// TwinCAT 3 PLC project PLC_PlantControl
// Title: PlantControl and CMs
// Company: ArmAutomation
// ProjectVersion: 0.1.0.0
// Description: This library hold functionality for a control structure and Control modules
// ProgramVersion: 3.1.4024.0
// libraries:
//   Tc2_ControllerToolbox, * (Beckhoff Automation GmbH)
//   Tc2_Standard, * (Beckhoff Automation GmbH)
//   Tc2_System, * (Beckhoff Automation GmbH)
//   Tc3_Module, * (Beckhoff Automation GmbH)
// project tree:
//   DUTs/Control Function UDTs/ ENUM_MODE_HANDLER.TcDUT
//   DUTs/V1/ Udt_CM_Actuator2State.TcDUT, Udt_CM_Actuator3State.TcDUT (not stored), Udt_CM_ActuatorAnalog.TcDUT (not stored), Udt_CM_Sensor2State.TcDUT, Udt_CM_SensorAnalog.TcDUT, Udt_PlantControl.TcDUT, Udt_PlantControl_SCADA.TcDUT (not stored)
//   DUTs/V2/ Udt_CM_Actuator2State_V2.TcDUT, Udt_CM_AO_V2.TcDUT, Udt_CM_Actuator3State_V2.TcDUT
//   GVLs/ FIO.TcGVL, OPC.TcGVL
//   / PlcTask.TcTTO
//   POUs/CM/ CM_Actuator2State.TcPOU, CM_Actuator3State.TcPOU, CM_ActuatorAnalog.TcPOU, CM_Sensor2State.TcPOU, CM_SensorAnalog.TcPOU
//   POUs/CM_V2/ CM_Actuator2State_V2.TcPOU, CM_Actuator3State_V2.TcPOU, CM_AO_V2.TcPOU, CM_Sensor2State_V2.TcPOU, CM_SensorAnalog_V2.TcPOU
//   POUs/Control functions/ FB_MODE_HANDLER.TcPOU, FB_PID.TcPOU
//   POUs/EM/ EM_Tank.TcPOU
//   POUs/ MAIN.TcPOU
//   POUs/Plant Control/ FB_PlantControl.TcPOU, FB_PlantControl_V2.TcPOU
//   POUs/Scaling/ FB_ScaleIN_1.TcPOU, FB_ScaleOut_1.TcPOU
//   POUs/System/ FB_ScaleIN.TcPOU, FB_ScaleOut.TcPOU, systemTimeDelay.TcPOU, SystemTimeTick.TcPOU
//   Version/ Global_Version.TcGVL
// real-time tasks:
//   TASK PlcTask: cycle T#10ms, priority 20, ADS port 350

CONFIGURATION PLC_PlantControl
    RESOURCE PLC ON TwinCAT3
        TASK PlcTask(INTERVAL := T#10ms, PRIORITY := 20);
        PROGRAM MAIN WITH PlcTask : MAIN;
    END_RESOURCE
END_CONFIGURATION

// ---- DUTs/Control Function UDTs/ENUM_MODE_HANDLER.TcDUT
{attribute 'qualified_only'}
{attribute 'strict'}
TYPE ENUM_MODE_HANDLER :
(
    MODE_EMGSTOP := 0,
    MODE_AUTO := 1,
    MODE_MAN  := 2
);
END_TYPE

// ---- DUTs/V1/Udt_CM_Actuator2State.TcDUT
TYPE Udt_CM_Actuator2State :
STRUCT
	PI_MANUAL :BOOL;
	PI_AUTO : BOOL;
	PI_HMI_HAND : BOOL;
	
	PI_AlarmHigh_Enable : BOOL;
	PI_AlarmLow_Enable : BOOL;
	
	PI_Alarm_Ack_H : BOOL;
	PI_Alarm_Ack_L : BOOL;
	
	PI_Interlock : BOOL;
	PO_Interlocked : BOOL;
	
	PO_ALARM_H : BOOL;
	PO_ALARM_L : BOOL;
	
	PO_HMI_HAND_ON: BOOL;
	PO_AUTO_ON : BOOL;
	PO_MANUAL_ON : BOOL;
	PO_ON : BOOL;
	PO_OFF :BOOL;
	
	
END_STRUCT
END_TYPE

// ---- DUTs/V1/Udt_CM_Sensor2State.TcDUT
TYPE Udt_CM_Sensor2State :
STRUCT
	PI_ManualMode : BOOL;
	PI_AutoHigh : BOOL;
	
	PI_HMI_HAND : BOOL;
	PI_HMI_HAND_ON : BOOL;
	
	PI_AlarmHighEnable : BOOL;
	PI_AlarmLowEnable : BOOL;
	
	PI_Alarmdelay_H : INT;
	PI_Alarmdelay_L : INT;
	
	PO_Alarm_H : BOOL;
	PO_Alarm_L : BOOL;
	
	PO_HMI_HAND : BOOL;
	PO_High : BOOL;
	
	PO_HIST_BIT_H : BOOL;
	PO_HIST_BIT_L : BOOL;

END_STRUCT
END_TYPE

// ---- DUTs/V1/Udt_CM_SensorAnalog.TcDUT
TYPE Udt_CM_SensorAnalog :
STRUCT
	PI_ManualMode : BOOL;
	PI_AutoMode : BOOL;
	
	PI_AlarmHighEnable : BOOL;
	PI_AlarmLowEnable : BOOL;
	PI_AlarmHighHighEnable : BOOL;
	PI_AlarmLowLowEnable : BOOL;
	
	PI_Alarm_Ack_HH : BOOL;
	PI_Alarm_Ack_H : BOOL;
	PI_Alarm_Ack_L : BOOL;
	PI_Alarm_Ack_LL : BOOL;
	
	
	PI_PV :INT;
	PI_PV_REAL : REAL;
	
	PI_PV_MAX : INT;
	PI_PV_MIN : INT;

	
	PO_PV_REAL : REAL;
	PO_PV_SCALED : REAL;
	
	
	PO_ALARM_HH : BOOL;
	PO_ALARM_H : BOOL;
	PO_ALARM_L : BOOL;
	PO_ALARM_LL : BOOL;
	
	PO_HIST_BIT_HH : BOOL;
	PO_HIST_BIT_H : BOOL;
	PO_HIST_BIT_L : BOOL;
	PO_HIST_BIT_LL : BOOL;
	
	
END_STRUCT
END_TYPE

// ---- DUTs/V1/Udt_PlantControl.TcDUT
TYPE Udt_PlantControl :
STRUCT
	
	PI_Auto : BOOL;
	PI_Manual : BOOL;
	
	
	PI_Start : BOOL;
	PI_Stop : BOOL := TRUE;
	PI_Reset : BOOL;
	PI_ResetEmgStop_5s :BOOL;
	
	PI_EmgStop : BOOL := TRUE;
	
	PO_Manual : BOOL;
	
	
	PO_Auto : BOOL;
	PO_Startet : BOOL;
	PO_Stopped : BOOL;
	PO_Reset : BOOL;
	PO_ResetEmgStop_5s :BOOL;
	
	PO_EmgStopped : BOOL;
	
	PO_ON : BOOL;
	
	PO_MODE : ENUM_MODE_HANDLER;
END_STRUCT
END_TYPE

// ---- DUTs/V2/Udt_CM_Actuator2State_V2.TcDUT
TYPE Udt_CM_Actuator2State_V2 :
STRUCT
	PI_MANUAL :BOOL;
	PI_AUTO : BOOL;
	PI_HMI_HAND : BOOL;
	
	PI_AlarmHigh_Enable : BOOL;
	PI_AlarmLow_Enable : BOOL;
	
	PI_Alarm_Condition_H : BOOL;
	PI_Alarm_Condition_L : BOOL;
	
	PI_AlarmDelay_H : LREAL;
	PI_AlarmDelay_L : LREAL;
	
	PI_Alarm_Ack_H : BOOL;
	PI_Alarm_Ack_L : BOOL;
	
	PI_Interlock : BOOL;
	(*PO_Interlocked : BOOL;
	
	PO_ALARM_H : BOOL;
	PO_ALARM_L : BOOL;
	
	PO_HMI_HAND_ON: BOOL;
	PO_AUTO_ON : BOOL;
	PO_MANUAL_ON : BOOL;
	PO_ON : BOOL;
	PO_OFF :BOOL;
	*)
	
	PO_MODE : ENUM_MODE_HANDLER;
	
END_STRUCT
END_TYPE

// ---- DUTs/V2/Udt_CM_AO_V2.TcDUT
TYPE Udt_CM_AO_V2 :
STRUCT
	PI_MANUAL :BOOL;
	PI_AUTO : BOOL;
	PI_HMI_HAND : BOOL; 
	
	PI_MANUAL_ON_1 : BOOL;
	PI_MANUAL_ON_2 : BOOL;
	
	PI_AUTO_ON_1 : BOOL;
	PI_AUTO_ON_2 : BOOL;
	
	PI_INTERLOCK : BOOL;
	
	PI_OFF : BOOL;
	
	PO_HMI_HAND_ON : BOOL;
	PO_AUTO_ON : BOOL;
	PO_ON : BOOL;
	
	
	PO_INTERLOCKED : BOOL;
	
	PO_OUT_OFF :BOOL;
	
	PI_Alarm_Ack_HH : BOOL;
	PI_Alarm_Ack_H : BOOL;
	PI_Alarm_Ack_L : BOOL;
	PI_Alarm_Ack_LL : BOOL;
	
	PO_MODE : ENUM_MODE_HANDLER;
END_STRUCT
END_TYPE

// ---- DUTs/V2/Udt_CM_Actuator3State_V2.TcDUT
TYPE Udt_CM_Actuator3State_V2 :
STRUCT
	PI_MANUAL :BOOL;
	PI_HMI_HAND : BOOL;
	PI_AUTO : BOOL;
	
	PI_MANUAL_ON_1 : BOOL;
	PI_MANUAL_ON_2 : BOOL;
	
	PI_AUTO_ON_1 : BOOL;
	PI_AUTO_ON_2 : BOOL;
	
	PI_OFF : BOOL;
	
	PI_Alarm_Enable : BOOL;
	PI_CM_Alarm : BOOL;
	
	PI_CM_Interlock : BOOL;
	
	PO_AUTO_ON :BOOL;
	PO_MANUAL_ON :BOOL;
	PO_HMI_HAND_ON : BOOL;
	
	PO_ON_1 : BOOL;
	PO_ON_2 : BOOL;
	
	PO_OFF :BOOL;
	
	PO_CM_Alarm : BOOL;
	
	PO_CM_Interlocked : BOOL;
	
	PO_MODE : ENUM_MODE_HANDLER;


END_STRUCT
END_TYPE

// ---- GVLs/FIO.TcGVL
{attribute 'qualified_only'}
VAR_GLOBAL
	
	(*bEmgStop : BOOL := TRUE; //Sensor	Bool	Emergency stop	0	TRUE
	bStart : BOOL;	//Sensor	Bool	Start	1	FALSE
	bStop : BOOL := TRUE;	//Sensor	Bool	Stop	3	TRUE
	bReset : BOOL;	//Sensor	Bool	Reset	4	FALSE
	bManual : BOOL;	//Sensor	Bool	Manual	5	TRUE
	bAuto : BOOL; 	//Sensor	Bool	Auto	6	FALSE
	
	bGreenLight : BOOL;
	bYellowLight : BOOL;
	bRedLight : BOOL;*)
		
	Plant_control : Udt_PlantControl;
	
END_VAR

// ---- GVLs/OPC.TcGVL
{attribute 'qualified_only'}
VAR_GLOBAL
	//cmActuator2State : Udt_CM_Actuator2State;
	Udt_PlantControl : Udt_PlantControl;
	
	Plant_1_Control : Udt_PlantControl;
END_VAR

// ---- Version/Global_Version.TcGVL
{attribute 'TcGenerated'}
{attribute 'no-analysis'}
{attribute 'linkalways'}
// This function has been automatically generated from the project information.
VAR_GLOBAL CONSTANT
	{attribute 'const_non_replaced'}
	stLibVersion_PlantControl_and_CMs : ST_LibVersion := (iMajor := 0, iMinor := 1, iBuild := 0, iRevision := 0, nFlags := 0, sVersion := '0.1.0.0');
END_VAR

// ---- POUs/MAIN.TcPOU
PROGRAM MAIN
VAR
	//Plant_Control : FB_PlantControl;
END_VAR
VAR_IN_OUT
	
END_VAR


(*fbPlantControl(
		//Set up variables to IO here
		
		(*Auto_In := HMI.bAuto,
		Manual_In := HMI.bManual,
		
		
		Start_In := HMI.bStart,
		Stop_In := HMI.bStop,
		EmgStop_In := HMI.bEmgStop,
		Reset_In := HMI.bReset,
		
		Startet_Out => HMI.bGreenLight,
		Stopped_Out => HMI.bYellowLight,
		EmgStopped_Out => HMI.bRedLight,*)
	
		Ctrl_Plant := FIO.Plant_control
		);
	
cmActuator2State(
	CM_UDT_CTRL := OPC.cmActuator2State,
	Plant_control := FIO.Plant_control
	);
	
	*)

END_PROGRAM

// ---- POUs/CM/CM_Actuator2State.TcPOU
FUNCTION_BLOCK CM_Actuator2State
VAR_INPUT
	CM_Number : INT;
	
	PI_MANUAL :BOOL;
	PI_AUTO : BOOL;
	
	PI_HMI_HAND : BOOL;
	
	PI_MANUAL_ON : BOOL;
	PI_AUTO_ON : BOOL;
	
	PI_OFF : BOOL;
	
	PI_AlarmHigh_Enable : BOOL;
	PI_AlarmLow_Enable : BOOL;
	PI_AlarmDelay_H : ULINT;
	PI_AlarmDelay_L : ULINT;
	
	PI_Alarm_Condition_H : BOOL;
	PI_Alarm_Condition_L : BOOL;
	
	PI_CM_Interlock : BOOL;
	
END_VAR
VAR_OUTPUT
	
	PO_AUTO_ON :BOOL;
	PO_MANUAL_ON : BOOL;
	PO_HMI_HAND_ON : BOOL;
	
	PO_OUT_ON : BOOL;
	OUT_OFF :BOOL;
	
	
	PO_ALARM_H : BOOL;
	PO_ALARM_L : BOOL;;
	
	PO_Interlocked : BOOL;
	
END_VAR
VAR
	SR_Auto: SR;
	SR_Manual : SR;
	
	Alarm_limit_Exceeded_H : BOOL;
	Alarm_limit_Exceeded_L : BOOL;
	
	Alarm_Ack_H : BOOL;
	Alarm_Ack_L : BOOL;
	
	alarmDelay_H : systemTimeDelay;
	alarmDelay_L : systemTimeDelay;
END_VAR
VAR_IN_OUT
	CM_UDT_CTRL : Udt_CM_Actuator2State;
END_VAR
VAR // added by the converter: edge detectors and wires of the graphical bodies
    _w1 : BOOL;
END_VAR

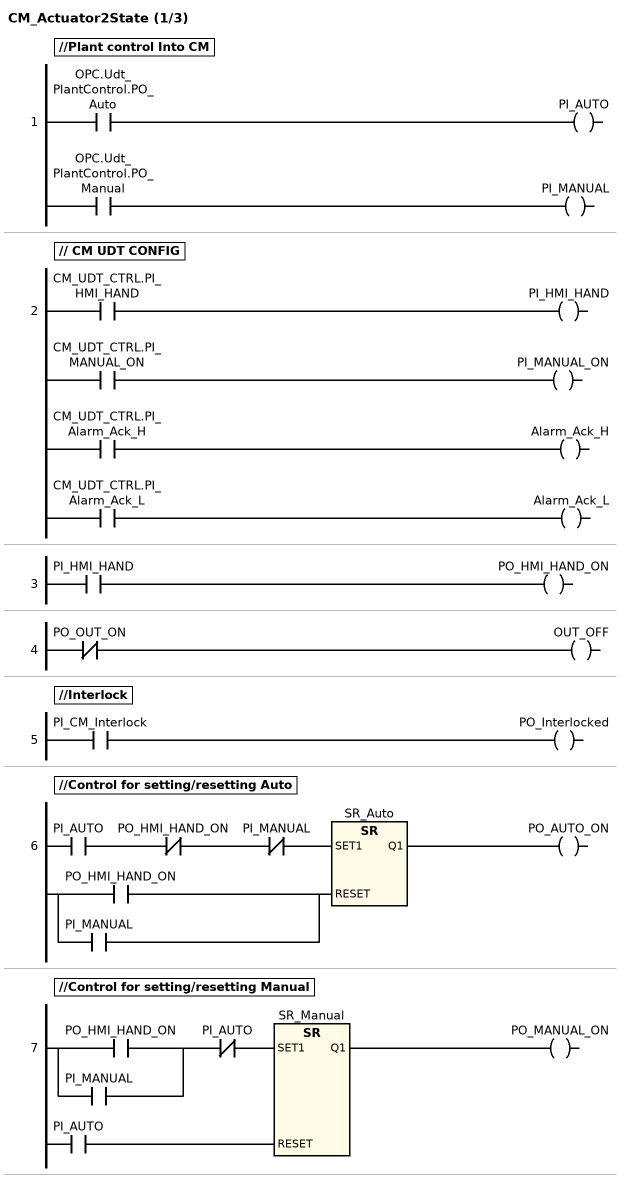
// NETWORK 1
// label: //Plant control Into CM
PI_AUTO := OPC.Udt_PlantControl.PO_Auto;
PI_MANUAL := OPC.Udt_PlantControl.PO_Manual;

// NETWORK 2
// label: // CM UDT CONFIG
PI_HMI_HAND := CM_UDT_CTRL.PI_HMI_HAND;
PI_MANUAL_ON := CM_UDT_CTRL.PI_MANUAL_ON;
Alarm_Ack_H := CM_UDT_CTRL.PI_Alarm_Ack_H;
Alarm_Ack_L := CM_UDT_CTRL.PI_Alarm_Ack_L;

// NETWORK 3
PO_HMI_HAND_ON := PI_HMI_HAND;

// NETWORK 4
OUT_OFF := NOT PO_OUT_ON;

// NETWORK 5
// label: //Interlock
PO_Interlocked := PI_CM_Interlock;

// NETWORK 6
// label: //Control for setting/resetting Auto
SR_Auto(SET1 := PI_AUTO AND NOT PO_HMI_HAND_ON AND NOT PI_MANUAL, RESET := PO_HMI_HAND_ON OR PI_MANUAL); // SR
PO_AUTO_ON := SR_Auto.Q1;

// NETWORK 7
// label: //Control for setting/resetting Manual
SR_Manual(SET1 := (PO_HMI_HAND_ON OR PI_MANUAL) AND NOT PI_AUTO, RESET := PI_AUTO); // SR
PO_MANUAL_ON := SR_Manual.Q1;

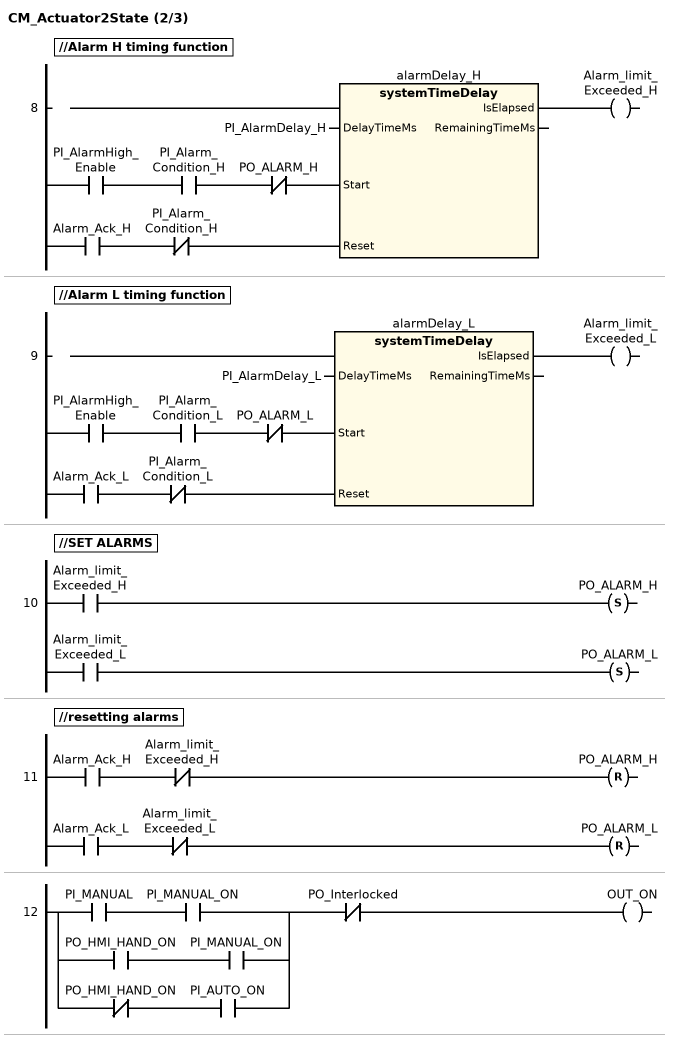
// NETWORK 8
// label: //Alarm H timing function
alarmDelay_H(
    DelayTimeMs := PI_AlarmDelay_H,
    Start := PI_AlarmHigh_Enable AND PI_Alarm_Condition_H AND NOT PO_ALARM_H,
    Reset := Alarm_Ack_H AND NOT PI_Alarm_Condition_H); // systemTimeDelay
Alarm_limit_Exceeded_H := alarmDelay_H.IsElapsed;

// NETWORK 9
// label: //Alarm L timing function
alarmDelay_L(
    DelayTimeMs := PI_AlarmDelay_L,
    Start := PI_AlarmHigh_Enable AND PI_Alarm_Condition_L AND NOT PO_ALARM_L,
    Reset := Alarm_Ack_L AND NOT PI_Alarm_Condition_L); // systemTimeDelay
Alarm_limit_Exceeded_L := alarmDelay_L.IsElapsed;

// NETWORK 10
// label: //SET ALARMS
PO_ALARM_H S= Alarm_limit_Exceeded_H;
PO_ALARM_L S= Alarm_limit_Exceeded_L;

// NETWORK 11
// label: //resetting alarms
PO_ALARM_H R= Alarm_Ack_H AND NOT Alarm_limit_Exceeded_H;
PO_ALARM_L R= Alarm_Ack_L AND NOT Alarm_limit_Exceeded_L;

// NETWORK 12
OUT_ON := (PI_MANUAL AND PI_MANUAL_ON OR PO_HMI_HAND_ON AND PI_MANUAL_ON OR NOT PO_HMI_HAND_ON AND PI_AUTO_ON) AND NOT PO_Interlocked;

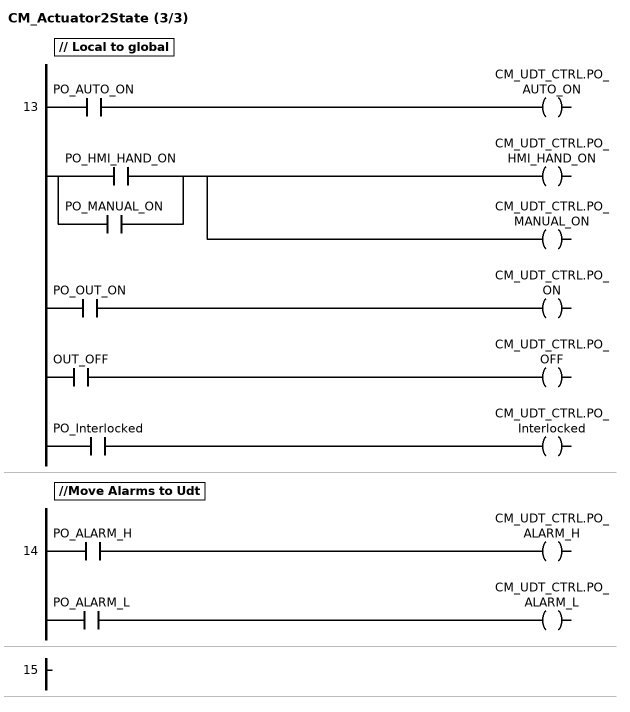
// NETWORK 13
// label: // Local to global
CM_UDT_CTRL.PO_AUTO_ON := PO_AUTO_ON;
_w1 := PO_HMI_HAND_ON OR PO_MANUAL_ON;
CM_UDT_CTRL.PO_HMI_HAND_ON := _w1;
CM_UDT_CTRL.PO_MANUAL_ON := _w1;
CM_UDT_CTRL.PO_ON := PO_OUT_ON;
CM_UDT_CTRL.PO_OFF := OUT_OFF;
CM_UDT_CTRL.PO_Interlocked := PO_Interlocked;

// NETWORK 14
// label: //Move Alarms to Udt
CM_UDT_CTRL.PO_ALARM_H := PO_ALARM_H;
CM_UDT_CTRL.PO_ALARM_L := PO_ALARM_L;

// NETWORK 15

END_FUNCTION_BLOCK

// ---- POUs/System/systemTimeDelay.TcPOU
FUNCTION_BLOCK systemTimeDelay
VAR_INPUT
    DelayTime : LREAL;   // Desired delay in seconds
    Start     : BOOL;    // Start signal (must stay TRUE to complete delay)
    Reset     : BOOL;    // Resets latched state and timer
END_VAR

VAR_OUTPUT
    IsElapsed     : BOOL;    // Latches TRUE after timeout, until reset
    RemainingTime : LREAL;   // Countdown in seconds (0 if not running)
END_VAR

VAR
    StartEdge       : BOOL;
    PrevStart       : BOOL;
    StartTime       : ULINT;   // Time when timer started (µs)
    ElapsedTimeRaw  : ULINT;   // Raw elapsed time in microseconds
    ElapsedSeconds  : LREAL;   // Elapsed time in seconds
    IsRunning       : BOOL;
END_VAR

// Detect rising edge of Start
StartEdge := Start AND NOT PrevStart;
PrevStart := Start;

// Reset everything if Reset = TRUE
IF Reset THEN
    IsElapsed := FALSE;
    IsRunning := FALSE;
    RemainingTime := 0.0;
END_IF

// If Start goes low during active timing, cancel and reset
IF NOT Start AND IsRunning THEN
    IsRunning := FALSE;
    RemainingTime := 0.0;
END_IF

// Start timer on rising edge of Start
IF StartEdge AND NOT IsElapsed THEN
    StartTime := F_GetSystemTime();  // System time in microseconds
    IsRunning := TRUE;
END_IF

// Timing logic
IF IsRunning THEN
    ElapsedTimeRaw := F_GetSystemTime() - StartTime;       // Time difference in µs
    ElapsedSeconds := ElapsedTimeRaw / 10000000.0;          // Convert to seconds

    IF ElapsedSeconds >= DelayTime THEN
        IsElapsed := TRUE;
        IsRunning := FALSE;
        RemainingTime := 0.0;
    ELSE
        RemainingTime := DelayTime - ElapsedSeconds;
    END_IF
END_IF

END_FUNCTION_BLOCK

// ---- POUs/CM/CM_Actuator3State.TcPOU
FUNCTION_BLOCK CM_Actuator3State
VAR_INPUT
	CM_Number : INT;
	
	IN_MANUAL :BOOL;
	IN_HMI_HAND : BOOL;
	IN_AUTO : BOOL;
	
	IN_MANUAL_ON_1 : BOOL;
	IN_MANUAL_ON_2 : BOOL;
	
	IN_AUTO_ON_1 : BOOL;
	IN_AUTO_ON_2 : BOOL;
	
	IN_OFF : BOOL;
	
	IN_Alarm_Enable : BOOL;
	IN_CM_Alarm : BOOL;
	
	IN_CM_Interlock : BOOL;
END_VAR
VAR_OUTPUT
	AUTO_ON :BOOL;
	HMI_HAND_ON : BOOL;
	
	OUT_ON_1 : BOOL;
	OUT_ON_2 : BOOL;
	
	OUT_OFF :BOOL;
	
	PO_CM_Alarm : BOOL;
	
	PO_CM_Interlocked : BOOL;
END_VAR
VAR
	alarmDelay_H : systemTimeDelay;
	alarmDelay_L : systemTimeDelay;
END_VAR
VAR_IN_OUT
	CM_UDT_CTRL : Udt_CM_Actuator3State;
	Plant_control : Udt_PlantControl;
END_VAR

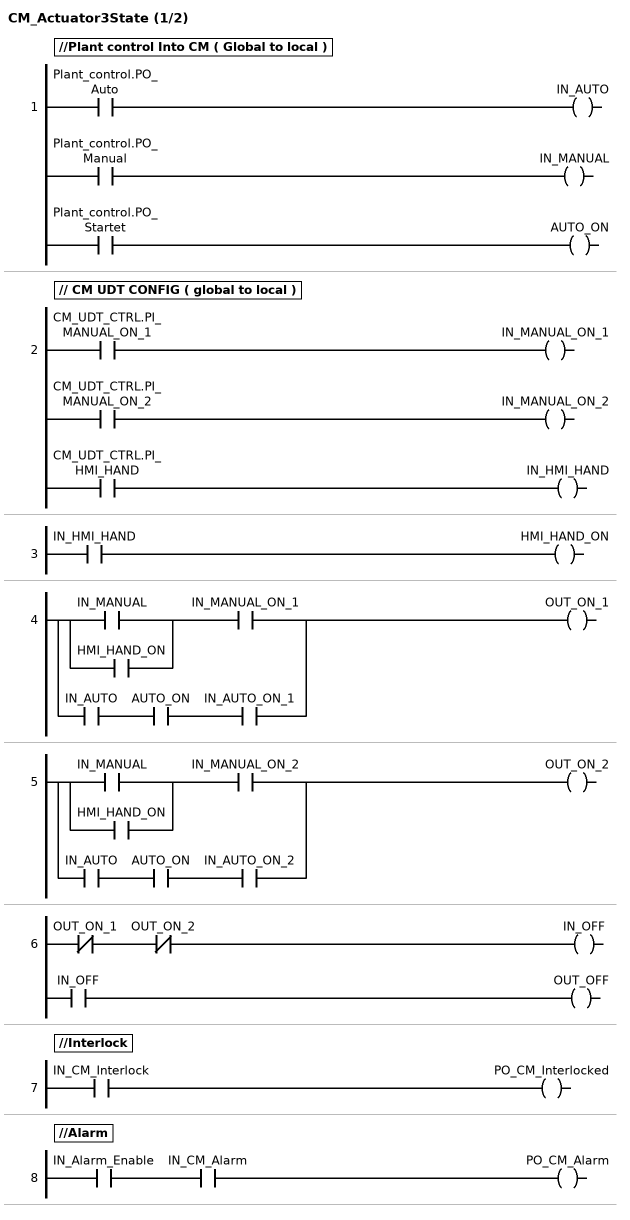
// NETWORK 1
// label: //Plant control Into CM ( Global to local )
IN_AUTO := Plant_control.PO_Auto;
IN_MANUAL := Plant_control.PO_Manual;
AUTO_ON := Plant_control.PO_Startet;

// NETWORK 2
// label: // CM UDT CONFIG ( global to local )
IN_MANUAL_ON_1 := CM_UDT_CTRL.PI_MANUAL_ON_1;
IN_MANUAL_ON_2 := CM_UDT_CTRL.PI_MANUAL_ON_2;
IN_HMI_HAND := CM_UDT_CTRL.PI_HMI_HAND;

// NETWORK 3
HMI_HAND_ON := IN_HMI_HAND;

// NETWORK 4
OUT_ON_1 := (IN_MANUAL OR HMI_HAND_ON) AND IN_MANUAL_ON_1 OR IN_AUTO AND AUTO_ON AND IN_AUTO_ON_1;

// NETWORK 5
OUT_ON_2 := (IN_MANUAL OR HMI_HAND_ON) AND IN_MANUAL_ON_2 OR IN_AUTO AND AUTO_ON AND IN_AUTO_ON_2;

// NETWORK 6
IN_OFF := NOT OUT_ON_1 AND NOT OUT_ON_2;
OUT_OFF := IN_OFF;

// NETWORK 7
// label: //Interlock
PO_CM_Interlocked := IN_CM_Interlock;

// NETWORK 8
// label: //Alarm
PO_CM_Alarm := IN_Alarm_Enable AND IN_CM_Alarm;

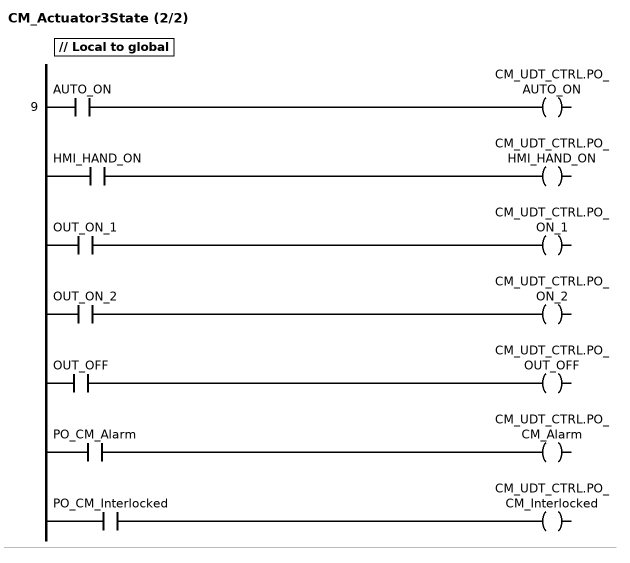
// NETWORK 9
// label: // Local to global
CM_UDT_CTRL.PO_AUTO_ON := AUTO_ON;
CM_UDT_CTRL.PO_HMI_HAND_ON := HMI_HAND_ON;
CM_UDT_CTRL.PO_ON_1 := OUT_ON_1;
CM_UDT_CTRL.PO_ON_2 := OUT_ON_2;
CM_UDT_CTRL.PO_OUT_OFF := OUT_OFF;
CM_UDT_CTRL.PO_CM_Alarm := PO_CM_Alarm;
CM_UDT_CTRL.PO_CM_Interlocked := PO_CM_Interlocked;

END_FUNCTION_BLOCK

// ---- POUs/CM/CM_ActuatorAnalog.TcPOU
FUNCTION_BLOCK CM_ActuatorAnalog
VAR_INPUT
	IN_MANUAL : BOOL;
	IN_AUTO : BOOL;
	IN_HMI_HAND : BOOL;
	
	IN_ON : BOOL;
	IN_OFF : BOOL;
	IN_EMG_STOP : BOOL;
	
	IN_RESET : BOOL;
	
	Input_analog : REAL;
	
	PV : REAL;
END_VAR
VAR_OUTPUT
	HMI_HAND_ON : BOOL;
	output_analog : REAL;
	Output_FB : BOOL;
END_VAR
VAR_IN_OUT
	CM_UDT_CTRL : Udt_CM_ActuatorAnalog;
	Plant_control : Udt_PlantControl;
END_VAR
VAR // added by the converter: edge detectors and wires of the graphical bodies
    _w1 : BOOL;
END_VAR

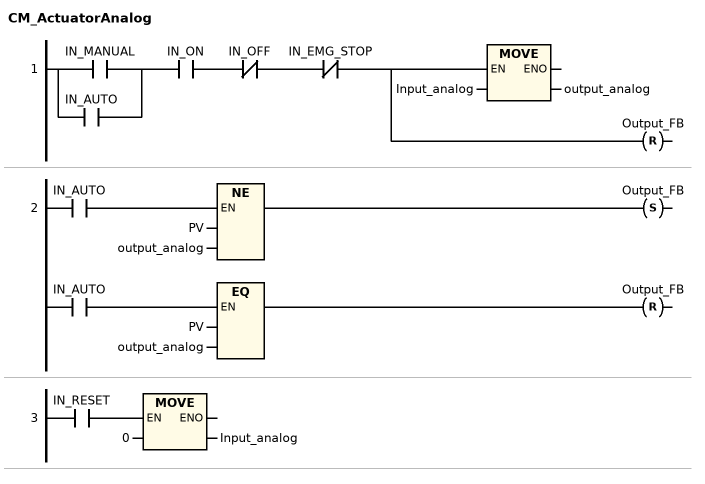
// NETWORK 1
_w1 := (IN_MANUAL OR IN_AUTO) AND IN_ON AND NOT IN_OFF AND NOT IN_EMG_STOP;
IF _w1 THEN output_analog := Input_analog; END_IF
Output_FB R= _w1;

// NETWORK 2
Output_FB S= IN_AUTO AND PV <> output_analog;
Output_FB R= IN_AUTO AND PV = output_analog;

// NETWORK 3
IF IN_RESET THEN Input_analog := 0; END_IF

END_FUNCTION_BLOCK

// ---- POUs/CM/CM_Sensor2State.TcPOU
FUNCTION_BLOCK CM_Sensor2State
VAR_INPUT
	PI_ManualMode : BOOL;
	PI_AutoMode : BOOL;
	
	PI_HMI_HAND : BOOL;
	PI_HMI_HAND_ON : BOOL;
	
	PI_Manual_ON : BOOL;
	PI_AutoHigh : BOOL;
	
	PI_AlarmHighEnable : BOOL;
	PI_AlarmLowEnable : BOOL;
	PI_Alarmdelay_H : DINT;
	PI_Alarmdelay_L : DINT;
	
	PI_Alarm_Condition_H : BOOL;
	PI_Alarm_Condition_L : BOOL;
	
	
	
END_VAR
VAR_OUTPUT
	PO_HMI_HAND : BOOL;
	PO_Manual : BOOL;
	PO_High : BOOL;
	
	PO_Alarm_H : BOOL;
	PO_Alarm_L : BOOL;
END_VAR
VAR
	Alarm_limit_Exceeded_H : BOOL;
	Alarm_limit_Exceeded_L : BOOL;
	
	prg_scan_H : DINT; // used for alarm delay
	prg_scan_L : DINT; // used for alarm delay
	
	Alarm_Ack_H : BOOL;
	Alarm_Ack_L : BOOL;
	
	alarmDelay_H : systemTimeDelay;
	alarmDelay_L : systemTimeDelay;
END_VAR
VAR_IN_OUT
	CM_UDT_CTRL : Udt_CM_Sensor2State;
	Plant_control : Udt_PlantControl;
END_VAR
VAR // added by the converter: edge detectors and wires of the graphical bodies
    _w1, _w2 : BOOL;
END_VAR

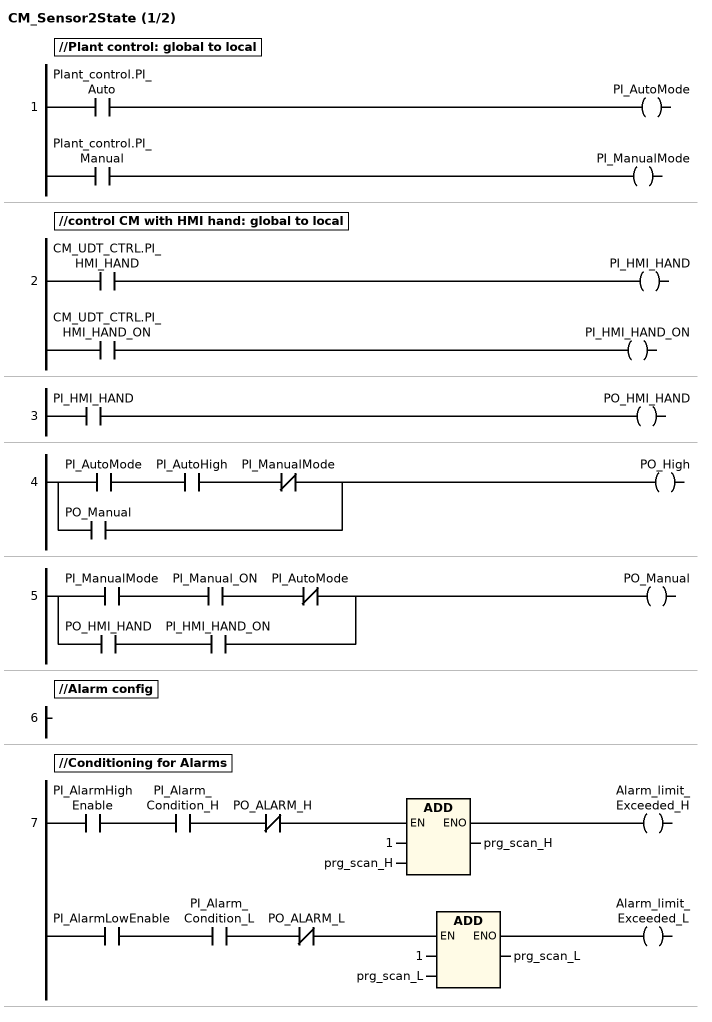
// NETWORK 1
// label: //Plant control: global to local
PI_AutoMode := Plant_control.PI_Auto;
PI_ManualMode := Plant_control.PI_Manual;

// NETWORK 2
// label: //control CM with HMI hand: global to local
PI_HMI_HAND := CM_UDT_CTRL.PI_HMI_HAND;
PI_HMI_HAND_ON := CM_UDT_CTRL.PI_HMI_HAND_ON;

// NETWORK 3
PO_HMI_HAND := PI_HMI_HAND;

// NETWORK 4
PO_High := PI_AutoMode AND PI_AutoHigh AND NOT PI_ManualMode OR PO_Manual;

// NETWORK 5
PO_Manual := PI_ManualMode AND PI_Manual_ON AND NOT PI_AutoMode OR PO_HMI_HAND AND PI_HMI_HAND_ON;

// NETWORK 6
// label: //Alarm config

// NETWORK 7
// label: //Conditioning for Alarms
_w1 := PI_AlarmHighEnable AND PI_Alarm_Condition_H AND NOT PO_ALARM_H;
IF _w1 THEN prg_scan_H := 1 + prg_scan_H; END_IF
Alarm_limit_Exceeded_H := _w1;
_w2 := PI_AlarmLowEnable AND PI_Alarm_Condition_L AND NOT PO_ALARM_L;
IF _w2 THEN prg_scan_L := 1 + prg_scan_L; END_IF
Alarm_limit_Exceeded_L := _w2;

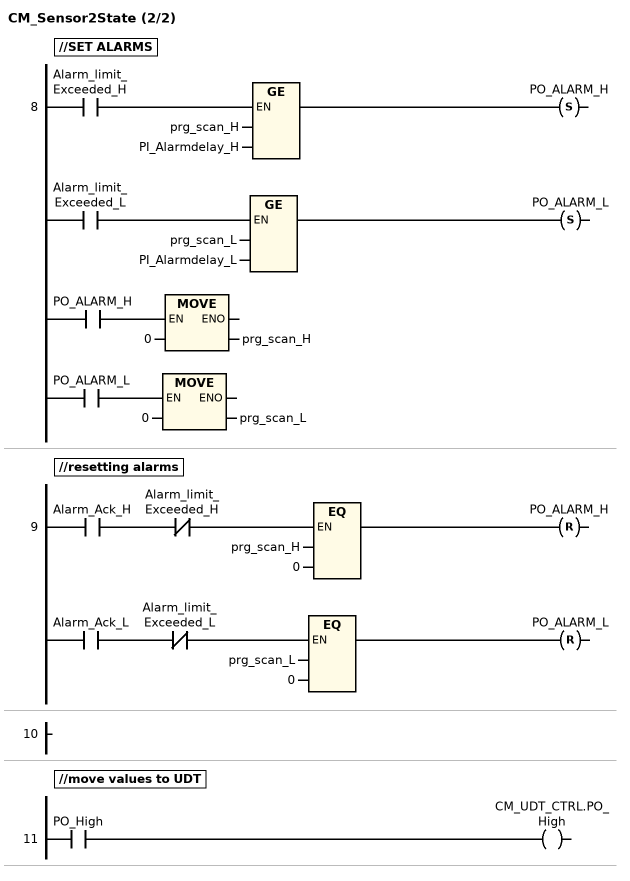
// NETWORK 8
// label: //SET ALARMS
PO_ALARM_H S= Alarm_limit_Exceeded_H AND prg_scan_H >= PI_Alarmdelay_H;
PO_ALARM_L S= Alarm_limit_Exceeded_L AND prg_scan_L >= PI_Alarmdelay_L;
IF PO_ALARM_H THEN prg_scan_H := 0; END_IF
IF PO_ALARM_L THEN prg_scan_L := 0; END_IF

// NETWORK 9
// label: //resetting alarms
PO_ALARM_H R= Alarm_Ack_H AND NOT Alarm_limit_Exceeded_H AND prg_scan_H = 0;
PO_ALARM_L R= Alarm_Ack_L AND NOT Alarm_limit_Exceeded_L AND prg_scan_L = 0;

// NETWORK 10

// NETWORK 11
// label: //move values to UDT
CM_UDT_CTRL.PO_High := PO_High;

END_FUNCTION_BLOCK

// ---- POUs/CM/CM_SensorAnalog.TcPOU
FUNCTION_BLOCK CM_SensorAnalog
VAR_INPUT
	
	PI_ManualMode : BOOL;
	PI_AutoMode : BOOL;
	
	//ALARMS:
	PI_AlarmHighHighEnable : BOOL;
	PI_AlarmHighEnable : BOOL;
	PI_AlarmLowEnable : BOOL;
	PI_AlarmLowLowEnable : BOOL;
	
	PI_AlarmHighHighLimit : REAL;
	PI_AlarmHighLimit : REAL;
	PI_AlarmLowLimit : REAL;
	PI_AlarmLowLowLimit : REAL;
	
	PI_AlarmDelay_HH : ULINT;
	PI_AlarmDelay_H : ULINT;
	PI_AlarmDelay_L : ULINT;
	PI_AlarmDelay_LL : ULINT;
	
	PI_PV :DINT;
	PI_PV_REAL : REAL;
	PI_PV_MANUAL : REAL;
	
	ENABLE_SCALING : BOOL;
	PI_PV_MAX_IN : INT;
	PI_PV_MIN_IN : INT;
	PI_PV_MAX_OUT : INT;
	PI_PV_MIN_OUT : INT;
END_VAR
VAR_OUTPUT
	
	PO_PV_SCALED : REAL;
	PO_PV_REAL : REAL;

	PO_ALARM_HH : BOOL;
	PO_ALARM_H : BOOL;
	PO_ALARM_L : BOOL;
	PO_ALARM_LL : BOOL;
END_VAR
VAR
	scale : Tc2_ControllerToolbox.FB_CTRL_SCALE;
	scaleParams : ST_CTRL_SCALE_PARAMS;
	
	Alarm_limit_Exceeded_HH : BOOL;
	Alarm_limit_Exceeded_H : BOOL;
	Alarm_limit_Exceeded_L : BOOL;
	Alarm_limit_Exceeded_LL : BOOL;
	
	Alarm_Ack_HH : BOOL;
	Alarm_Ack_H : BOOL;
	Alarm_Ack_L : BOOL;
	Alarm_Ack_LL : BOOL;
	
	alarmDelay_HH : systemTimeDelay;
	alarmDelay_H : systemTimeDelay;
	alarmDelay_L : systemTimeDelay;
	alarmDelay_LL : systemTimeDelay;
	
END_VAR
VAR_IN_OUT
	CM_UDT_CTRL : Udt_CM_SensorAnalog;
	Plant_control : Udt_PlantControl;
END_VAR

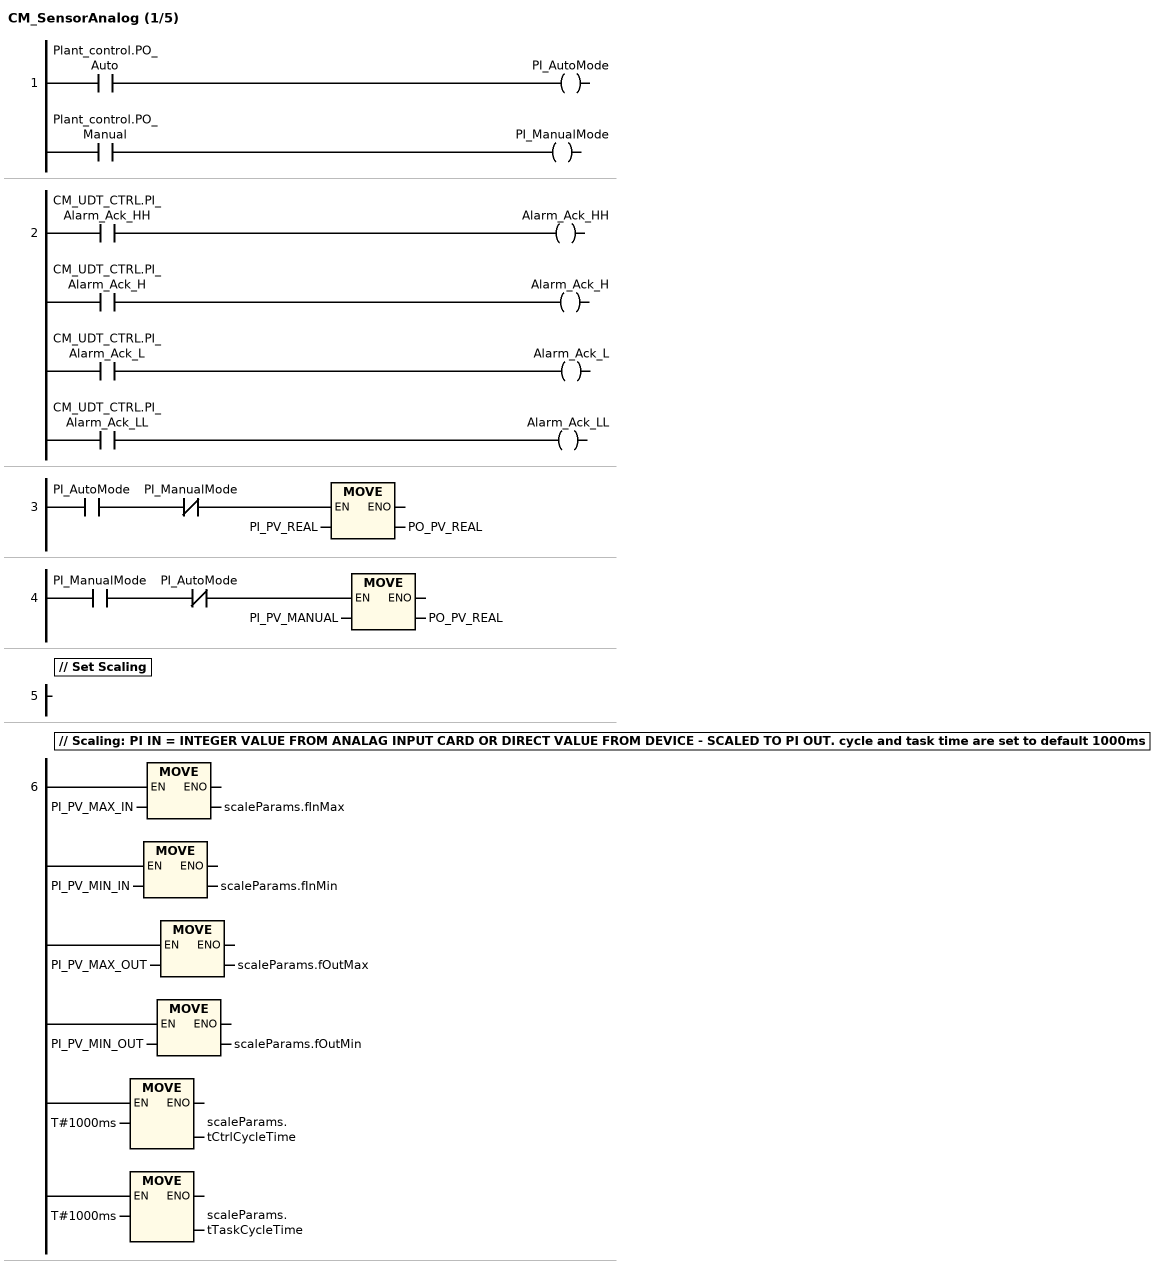
// NETWORK 1
PI_AutoMode := Plant_control.PO_Auto;
PI_ManualMode := Plant_control.PO_Manual;

// NETWORK 2
Alarm_Ack_HH := CM_UDT_CTRL.PI_Alarm_Ack_HH;
Alarm_Ack_H := CM_UDT_CTRL.PI_Alarm_Ack_H;
Alarm_Ack_L := CM_UDT_CTRL.PI_Alarm_Ack_L;
Alarm_Ack_LL := CM_UDT_CTRL.PI_Alarm_Ack_LL;

// NETWORK 3
IF PI_AutoMode AND NOT PI_ManualMode THEN PO_PV_REAL := PI_PV_REAL; END_IF

// NETWORK 4
IF PI_ManualMode AND NOT PI_AutoMode THEN PO_PV_REAL := PI_PV_MANUAL; END_IF

// NETWORK 5
// label: // Set Scaling

// NETWORK 6
// label: // Scaling: PI IN = INTEGER VALUE FROM ANALAG INPUT CARD OR DIRECT VALUE FROM DEVICE - SCALED TO PI OUT. cycle and task time are set to default 1000ms
scaleParams.fInMax := PI_PV_MAX_IN;
scaleParams.fInMin := PI_PV_MIN_IN;
scaleParams.fOutMax := PI_PV_MAX_OUT;
scaleParams.fOutMin := PI_PV_MIN_OUT;
scaleParams.tCtrlCycleTime := T#1000ms;
scaleParams.tTaskCycleTime := T#1000ms;

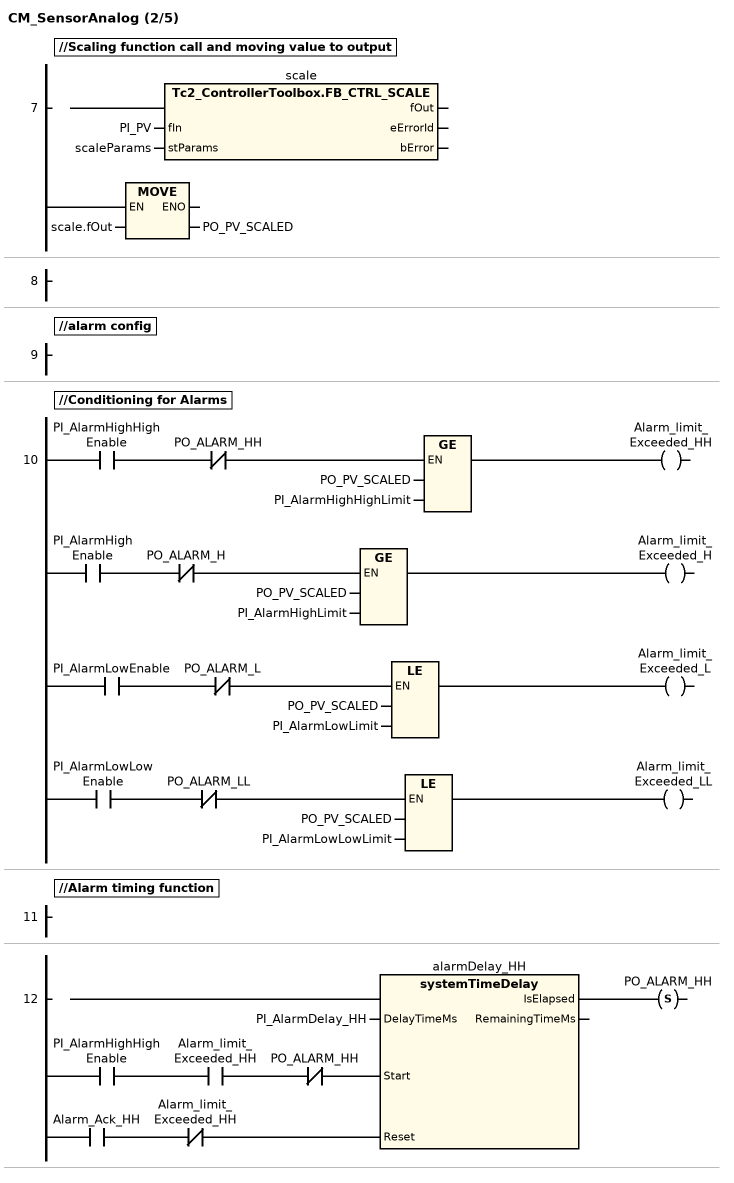
// NETWORK 7
// label: //Scaling function call and moving value to output
scale(fIn := PI_PV, stParams := scaleParams); // Tc2_ControllerToolbox.FB_CTRL_SCALE
PO_PV_SCALED := scale.fOut;

// NETWORK 8

// NETWORK 9
// label: //alarm config

// NETWORK 10
// label: //Conditioning for Alarms
Alarm_limit_Exceeded_HH := PI_AlarmHighHighEnable AND NOT PO_ALARM_HH AND PO_PV_SCALED >= PI_AlarmHighHighLimit;
Alarm_limit_Exceeded_H := PI_AlarmHighEnable AND NOT PO_ALARM_H AND PO_PV_SCALED >= PI_AlarmHighLimit;
Alarm_limit_Exceeded_L := PI_AlarmLowEnable AND NOT PO_ALARM_L AND PO_PV_SCALED <= PI_AlarmLowLimit;
Alarm_limit_Exceeded_LL := PI_AlarmLowLowEnable AND NOT PO_ALARM_LL AND PO_PV_SCALED <= PI_AlarmLowLowLimit;

// NETWORK 11
// label: //Alarm timing function

// NETWORK 12
alarmDelay_HH(
    DelayTimeMs := PI_AlarmDelay_HH,
    Start := PI_AlarmHighHighEnable AND Alarm_limit_Exceeded_HH AND NOT PO_ALARM_HH,
    Reset := Alarm_Ack_HH AND NOT Alarm_limit_Exceeded_HH); // systemTimeDelay
PO_ALARM_HH S= alarmDelay_HH.IsElapsed;

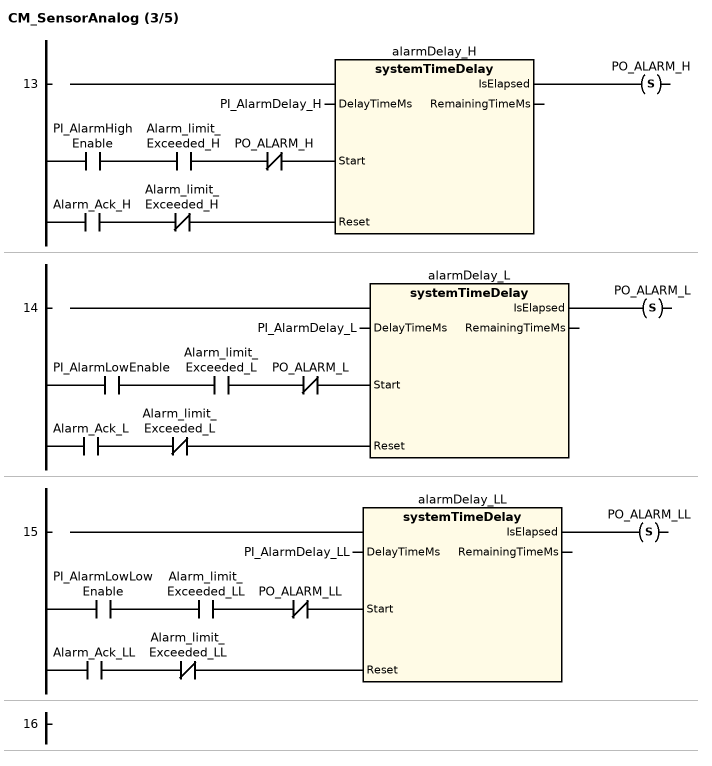
// NETWORK 13
alarmDelay_H(
    DelayTimeMs := PI_AlarmDelay_H,
    Start := PI_AlarmHighEnable AND Alarm_limit_Exceeded_H AND NOT PO_ALARM_H,
    Reset := Alarm_Ack_H AND NOT Alarm_limit_Exceeded_H); // systemTimeDelay
PO_ALARM_H S= alarmDelay_H.IsElapsed;

// NETWORK 14
alarmDelay_L(
    DelayTimeMs := PI_AlarmDelay_L,
    Start := PI_AlarmLowEnable AND Alarm_limit_Exceeded_L AND NOT PO_ALARM_L,
    Reset := Alarm_Ack_L AND NOT Alarm_limit_Exceeded_L); // systemTimeDelay
PO_ALARM_L S= alarmDelay_L.IsElapsed;

// NETWORK 15
alarmDelay_LL(
    DelayTimeMs := PI_AlarmDelay_LL,
    Start := PI_AlarmLowLowEnable AND Alarm_limit_Exceeded_LL AND NOT PO_ALARM_LL,
    Reset := Alarm_Ack_LL AND NOT Alarm_limit_Exceeded_LL); // systemTimeDelay
PO_ALARM_LL S= alarmDelay_LL.IsElapsed;

// NETWORK 16

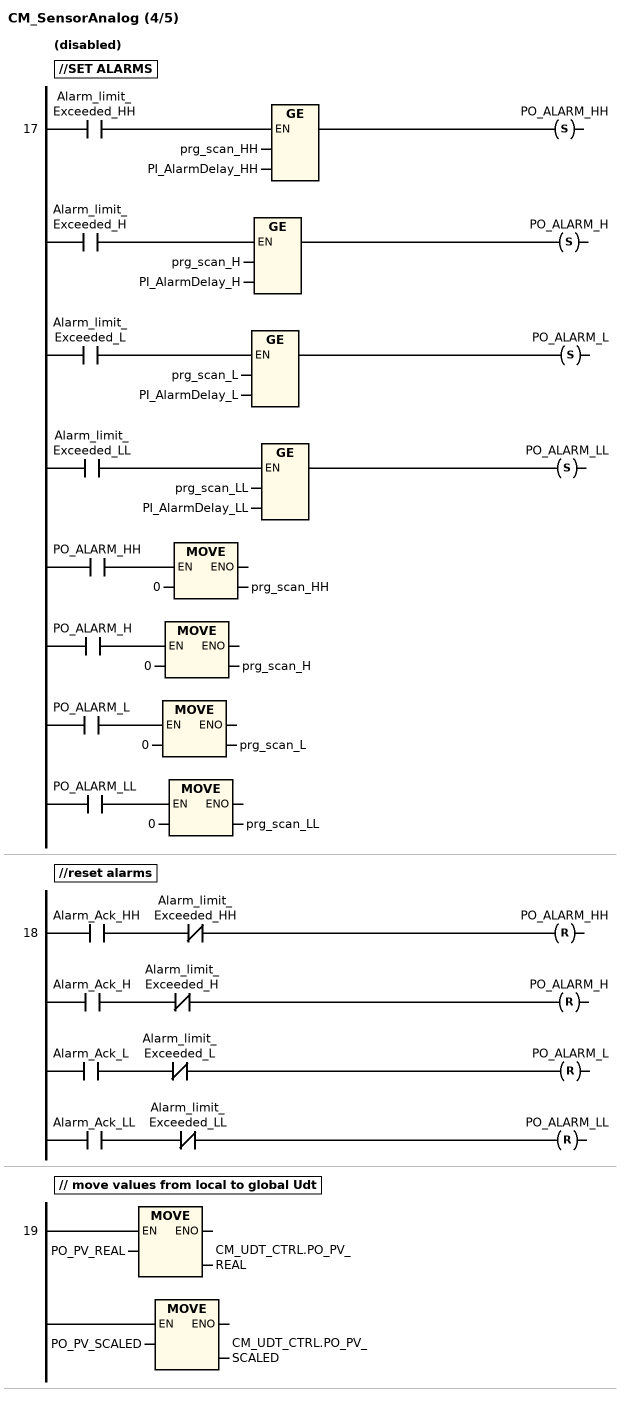
// NETWORK 17 (disabled)
// label: //SET ALARMS
// PO_ALARM_HH S= Alarm_limit_Exceeded_HH AND prg_scan_HH >= PI_AlarmDelay_HH;
// PO_ALARM_H S= Alarm_limit_Exceeded_H AND prg_scan_H >= PI_AlarmDelay_H;
// PO_ALARM_L S= Alarm_limit_Exceeded_L AND prg_scan_L >= PI_AlarmDelay_L;
// PO_ALARM_LL S= Alarm_limit_Exceeded_LL AND prg_scan_LL >= PI_AlarmDelay_LL;
// IF PO_ALARM_HH THEN prg_scan_HH := 0; END_IF
// IF PO_ALARM_H THEN prg_scan_H := 0; END_IF
// IF PO_ALARM_L THEN prg_scan_L := 0; END_IF
// IF PO_ALARM_LL THEN prg_scan_LL := 0; END_IF

// NETWORK 18
// label: //reset alarms
PO_ALARM_HH R= Alarm_Ack_HH AND NOT Alarm_limit_Exceeded_HH;
PO_ALARM_H R= Alarm_Ack_H AND NOT Alarm_limit_Exceeded_H;
PO_ALARM_L R= Alarm_Ack_L AND NOT Alarm_limit_Exceeded_L;
PO_ALARM_LL R= Alarm_Ack_LL AND NOT Alarm_limit_Exceeded_LL;

// NETWORK 19
// label: // move values from local to global Udt
CM_UDT_CTRL.PO_PV_REAL := PO_PV_REAL;
CM_UDT_CTRL.PO_PV_SCALED := PO_PV_SCALED;

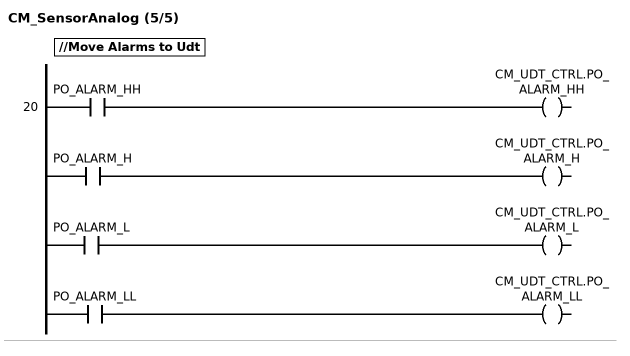
// NETWORK 20
// label: //Move Alarms to Udt
CM_UDT_CTRL.PO_ALARM_HH := PO_ALARM_HH;
CM_UDT_CTRL.PO_ALARM_H := PO_ALARM_H;
CM_UDT_CTRL.PO_ALARM_L := PO_ALARM_L;
CM_UDT_CTRL.PO_ALARM_LL := PO_ALARM_LL;

END_FUNCTION_BLOCK

// ---- POUs/CM_V2/CM_Actuator2State_V2.TcPOU
FUNCTION_BLOCK CM_Actuator2State_V2
VAR_INPUT
	
 	IN_ON : BOOL;
	Local_MODE_request : ENUM_MODE_HANDLER;
	Global_MODE_request : ENUM_MODE_HANDLER;
	
	PI_MANUAL :BOOL;
	PI_AUTO : BOOL;
	PI_HMI_HAND : BOOL;
	
	PI_AlarmHigh_Enable : BOOL;
	PI_AlarmLow_Enable : BOOL;
	
	PI_Alarm_Condition_H : BOOL;
	PI_Alarm_Condition_L : BOOL;
	
	PI_AlarmDelay_H : LREAL;
	PI_AlarmDelay_L : LREAL;
	
	PI_Alarm_Ack_H : BOOL;
	PI_Alarm_Ack_L : BOOL;
	
	PI_Interlock : BOOL;
	
	
	
END_VAR
VAR_OUTPUT
	PO_AUTO_ON :BOOL;
	PO_MANUAL_ON : BOOL;
	PO_HMI_HAND_ON : BOOL;
	
	PO_OUT_ON : BOOL;
	PO_OUT_OFF :BOOL;
	
	
	PO_ALARM_H : BOOL;
	PO_ALARM_L : BOOL;;
	
	PO_Interlocked : BOOL;
	
END_VAR
VAR
	SR_Auto: SR;
	SR_Manual : SR;
	
	Alarm_limit_Exceeded_H : BOOL;
	Alarm_limit_Exceeded_L : BOOL;
	
	Alarm_Ack_H : BOOL;
	Alarm_Ack_L : BOOL;
	
	alarmDelay_H : systemTimeDelay;
	alarmDelay_L : systemTimeDelay;
	
	MODE_HANDLER : FB_MODE_HANDLER;
END_VAR
VAR_IN_OUT
END_VAR

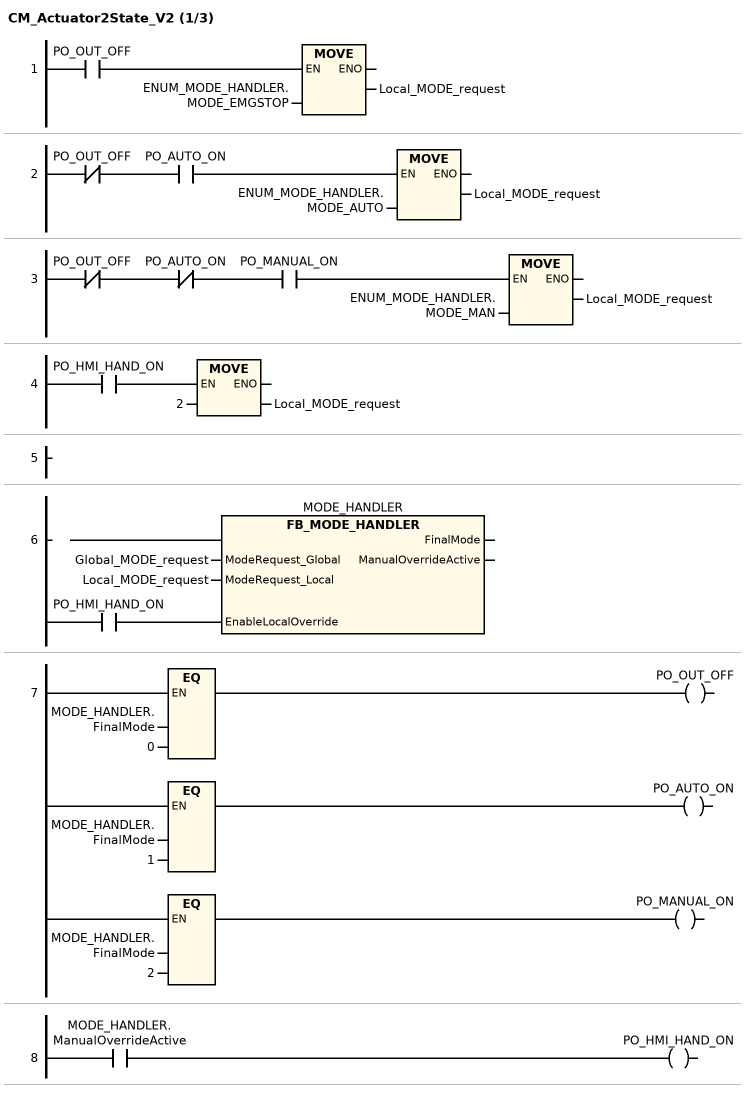
// NETWORK 1
IF PO_OUT_OFF THEN Local_MODE_request := ENUM_MODE_HANDLER.MODE_EMGSTOP; END_IF

// NETWORK 2
IF NOT PO_OUT_OFF AND PO_AUTO_ON THEN Local_MODE_request := ENUM_MODE_HANDLER.MODE_AUTO; END_IF

// NETWORK 3
IF NOT PO_OUT_OFF AND NOT PO_AUTO_ON AND PO_MANUAL_ON THEN Local_MODE_request := ENUM_MODE_HANDLER.MODE_MAN; END_IF

// NETWORK 4
IF PO_HMI_HAND_ON THEN Local_MODE_request := 2; END_IF

// NETWORK 5

// NETWORK 6
MODE_HANDLER(
    ModeRequest_Global := Global_MODE_request,
    ModeRequest_Local := Local_MODE_request,
    EnableLocalOverride := PO_HMI_HAND_ON); // FB_MODE_HANDLER

// NETWORK 7
PO_OUT_OFF := MODE_HANDLER.FinalMode = 0;
PO_AUTO_ON := MODE_HANDLER.FinalMode = 1;
PO_MANUAL_ON := MODE_HANDLER.FinalMode = 2;

// NETWORK 8
PO_HMI_HAND_ON := MODE_HANDLER.ManualOverrideActive;

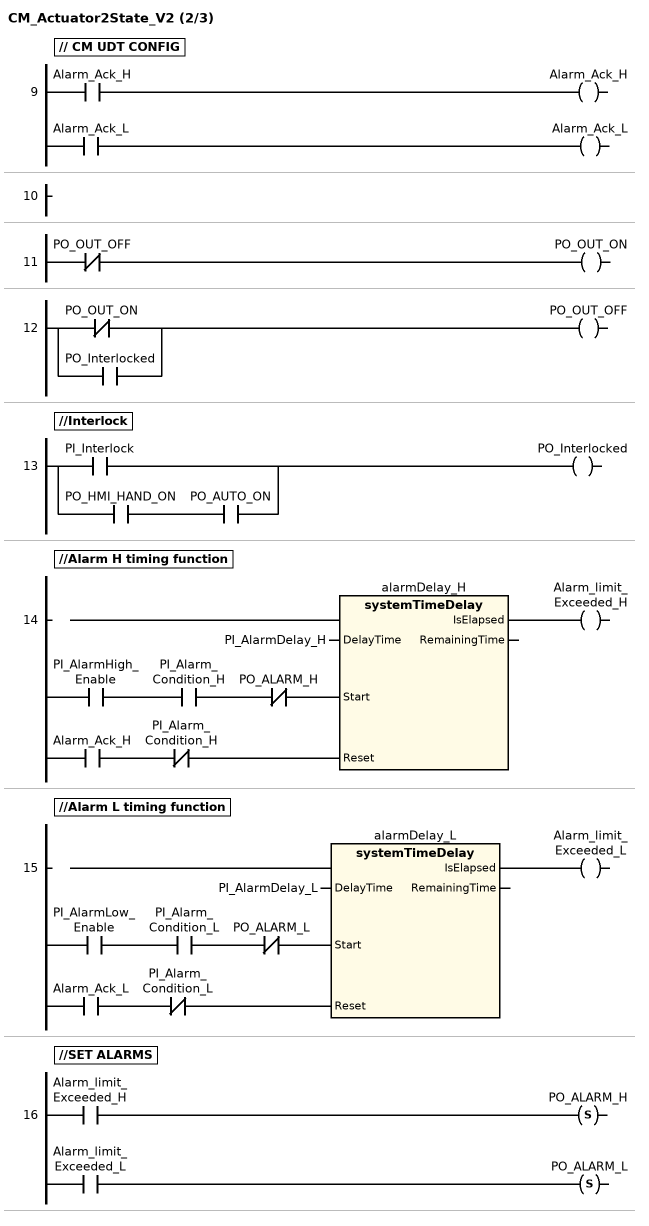
// NETWORK 9
// label: // CM UDT CONFIG
Alarm_Ack_H := Alarm_Ack_H;
Alarm_Ack_L := Alarm_Ack_L;

// NETWORK 10

// NETWORK 11
PO_OUT_ON := NOT PO_OUT_OFF;

// NETWORK 12
PO_OUT_OFF := NOT PO_OUT_ON OR PO_Interlocked;

// NETWORK 13
// label: //Interlock
PO_Interlocked := PI_Interlock OR PO_HMI_HAND_ON AND PO_AUTO_ON;

// NETWORK 14
// label: //Alarm H timing function
alarmDelay_H(
    DelayTime := PI_AlarmDelay_H,
    Start := PI_AlarmHigh_Enable AND PI_Alarm_Condition_H AND NOT PO_ALARM_H,
    Reset := Alarm_Ack_H AND NOT PI_Alarm_Condition_H); // systemTimeDelay
Alarm_limit_Exceeded_H := alarmDelay_H.IsElapsed;

// NETWORK 15
// label: //Alarm L timing function
alarmDelay_L(
    DelayTime := PI_AlarmDelay_L,
    Start := PI_AlarmLow_Enable AND PI_Alarm_Condition_L AND NOT PO_ALARM_L,
    Reset := Alarm_Ack_L AND NOT PI_Alarm_Condition_L); // systemTimeDelay
Alarm_limit_Exceeded_L := alarmDelay_L.IsElapsed;

// NETWORK 16
// label: //SET ALARMS
PO_ALARM_H S= Alarm_limit_Exceeded_H;
PO_ALARM_L S= Alarm_limit_Exceeded_L;

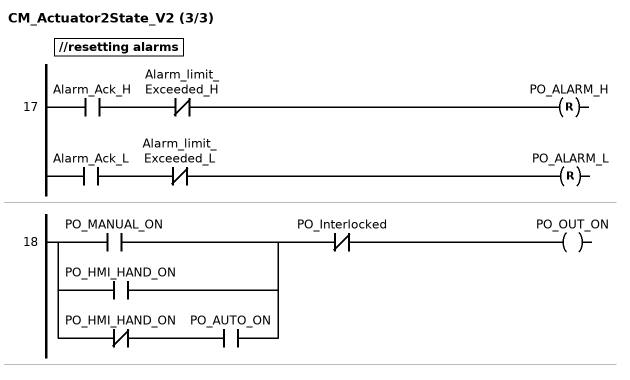
// NETWORK 17
// label: //resetting alarms
PO_ALARM_H R= Alarm_Ack_H AND NOT Alarm_limit_Exceeded_H;
PO_ALARM_L R= Alarm_Ack_L AND NOT Alarm_limit_Exceeded_L;

// NETWORK 18
PO_OUT_ON := (PO_MANUAL_ON OR PO_HMI_HAND_ON OR NOT PO_HMI_HAND_ON AND PO_AUTO_ON) AND NOT PO_Interlocked;

END_FUNCTION_BLOCK

// ---- POUs/Control functions/FB_MODE_HANDLER.TcPOU
FUNCTION_BLOCK FB_MODE_HANDLER
VAR_INPUT
	ModeRequest_Global : ENUM_MODE_HANDLER;
    ModeRequest_Local  : ENUM_MODE_HANDLER;
    EnableLocalOverride : BOOL := TRUE; // Optional
END_VAR
VAR_OUTPUT
	FinalMode : ENUM_MODE_HANDLER;
    ManualOverrideActive : BOOL;
END_VAR
VAR
END_VAR

 	(*
	MODE_EMGSTOP := 0,
    MODE_AUTO := 1,
    MODE_MAN  := 2
	*)

IF EnableLocalOverride AND (ModeRequest_Local = ENUM_MODE_HANDLER.MODE_MAN) THEN
    FinalMode := ENUM_MODE_HANDLER.MODE_MAN;
    ManualOverrideActive := TRUE;
ELSE
    FinalMode := ModeRequest_Global;
    ManualOverrideActive := FALSE;
END_IF;

// Safe fallback
IF (FinalMode <> ENUM_MODE_HANDLER.MODE_AUTO) AND 
   (FinalMode <> ENUM_MODE_HANDLER.MODE_MAN) THEN
    FinalMode := ENUM_MODE_HANDLER.MODE_EMGSTOP;
END_IF;

END_FUNCTION_BLOCK

// ---- POUs/CM_V2/CM_Actuator3State_V2.TcPOU
FUNCTION_BLOCK CM_Actuator3State_V2
VAR_INPUT
	Local_MODE_request : ENUM_MODE_HANDLER;
	Global_MODE_request : ENUM_MODE_HANDLER;
	
	PI_MANUAL :BOOL;
	PI_HMI_HAND : BOOL;
	PI_AUTO : BOOL;
	
	PI_MANUAL_ON_1 : BOOL;
	PI_MANUAL_ON_2 : BOOL;
	
	PI_AUTO_ON_1 : BOOL;
	PI_AUTO_ON_2 : BOOL;
	
	PI_OFF : BOOL;
	
	PI_Alarm_Enable : BOOL;
	PI_CM_Alarm : BOOL;
	
	PI_CM_Interlock : BOOL;
END_VAR
VAR_OUTPUT
	IN_ON : BOOL;
	
	PO_AUTO_ON :BOOL;
	PO_MANUAL_ON :BOOL;
	PO_HMI_HAND_ON : BOOL;
	
	PO_ON_1 : BOOL;
	PO_ON_2 : BOOL;
	
	PO_OFF :BOOL;
	
	PO_CM_Alarm : BOOL;
	
	PO_CM_Interlocked : BOOL;
	
	
END_VAR
VAR
	alarmDelay_H : systemTimeDelay;
	alarmDelay_L : systemTimeDelay;
	
	MODE_HANDLER : FB_MODE_HANDLER;
END_VAR
VAR_IN_OUT
	
END_VAR

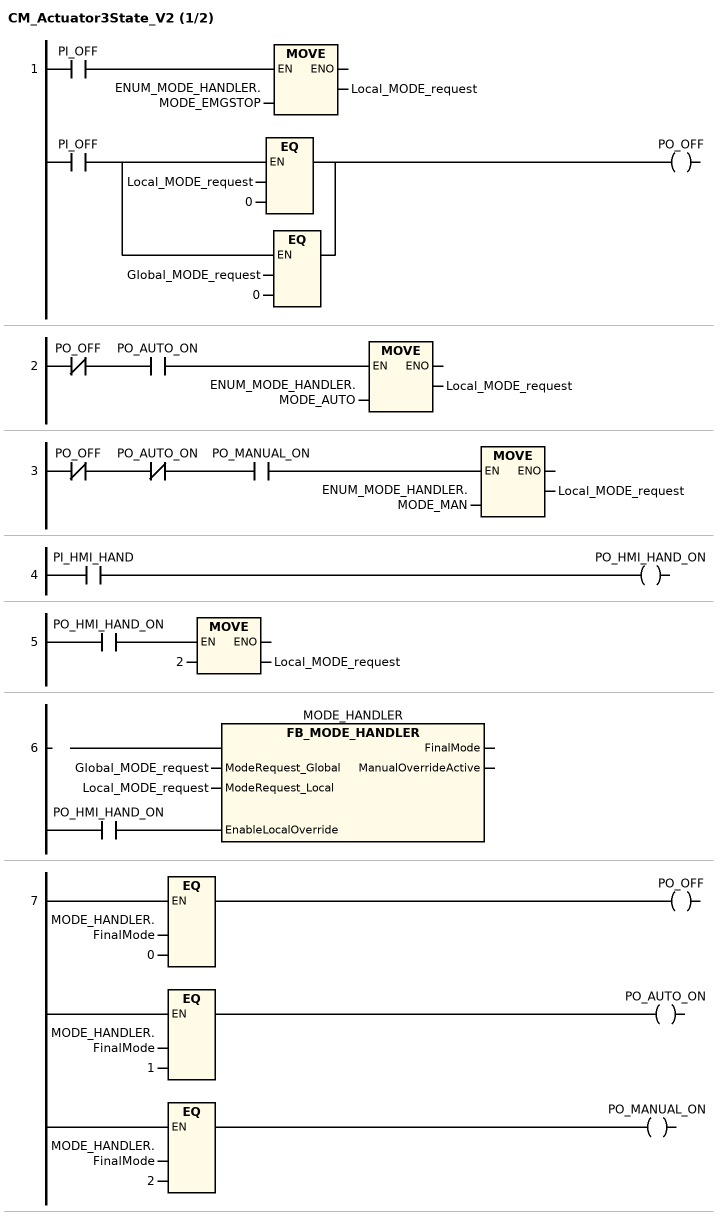
// NETWORK 1
IF PI_OFF THEN Local_MODE_request := ENUM_MODE_HANDLER.MODE_EMGSTOP; END_IF
PO_OFF := PI_OFF AND Local_MODE_request = 0 OR PI_OFF AND Global_MODE_request = 0;

// NETWORK 2
IF NOT PO_OFF AND PO_AUTO_ON THEN Local_MODE_request := ENUM_MODE_HANDLER.MODE_AUTO; END_IF

// NETWORK 3
IF NOT PO_OFF AND NOT PO_AUTO_ON AND PO_MANUAL_ON THEN Local_MODE_request := ENUM_MODE_HANDLER.MODE_MAN; END_IF

// NETWORK 4
PO_HMI_HAND_ON := PI_HMI_HAND;

// NETWORK 5
IF PO_HMI_HAND_ON THEN Local_MODE_request := 2; END_IF

// NETWORK 6
MODE_HANDLER(
    ModeRequest_Global := Global_MODE_request,
    ModeRequest_Local := Local_MODE_request,
    EnableLocalOverride := PO_HMI_HAND_ON); // FB_MODE_HANDLER

// NETWORK 7
PO_OFF := MODE_HANDLER.FinalMode = 0;
PO_AUTO_ON := MODE_HANDLER.FinalMode = 1;
PO_MANUAL_ON := MODE_HANDLER.FinalMode = 2;

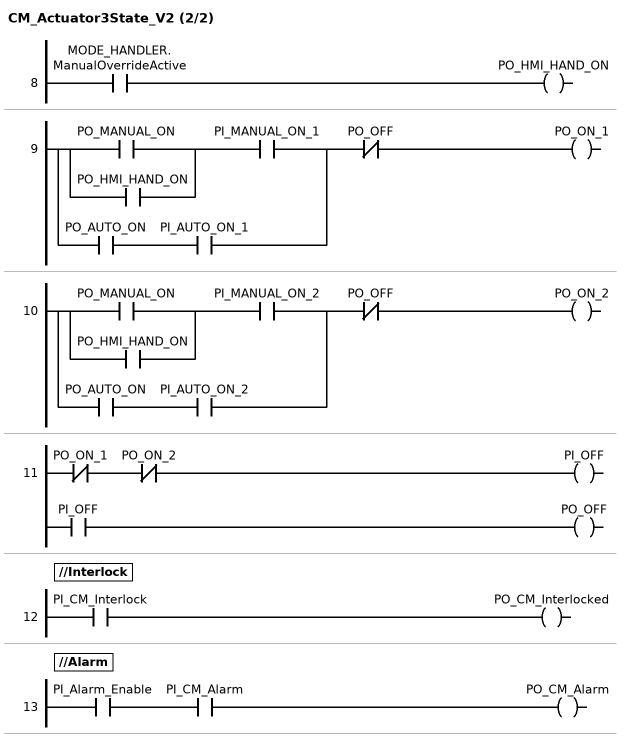
// NETWORK 8
PO_HMI_HAND_ON := MODE_HANDLER.ManualOverrideActive;

// NETWORK 9
PO_ON_1 := ((PO_MANUAL_ON OR PO_HMI_HAND_ON) AND PI_MANUAL_ON_1 OR PO_AUTO_ON AND PI_AUTO_ON_1) AND NOT PO_OFF;

// NETWORK 10
PO_ON_2 := ((PO_MANUAL_ON OR PO_HMI_HAND_ON) AND PI_MANUAL_ON_2 OR PO_AUTO_ON AND PI_AUTO_ON_2) AND NOT PO_OFF;

// NETWORK 11
PI_OFF := NOT PO_ON_1 AND NOT PO_ON_2;
PO_OFF := PI_OFF;

// NETWORK 12
// label: //Interlock
PO_CM_Interlocked := PI_CM_Interlock;

// NETWORK 13
// label: //Alarm
PO_CM_Alarm := PI_Alarm_Enable AND PI_CM_Alarm;

END_FUNCTION_BLOCK

// ---- POUs/CM_V2/CM_AO_V2.TcPOU
FUNCTION_BLOCK CM_AO_V2
VAR_INPUT
	IN_ON : BOOL;

	PI_PV : DINT; // Input from sensor or other device which should control
	
	SP_AUTO : DINT;
	SP_MAN: DINT;
	
	PI_HMI_HAND_ON :BOOL;
	
	
	Local_MODE_request : ENUM_MODE_HANDLER;
	Global_MODE_request : ENUM_MODE_HANDLER;
	
	
	//PID_PARAMS : ST_CTRL_PID_PARAMS;
	
	
	//ALARMS:
	PI_AlarmHighHighEnable : BOOL;
	PI_AlarmHighEnable : BOOL;
	PI_AlarmLowEnable : BOOL;
	PI_AlarmLowLowEnable : BOOL;
	
	PI_AlarmHighHighLimit : REAL;
	PI_AlarmHighLimit : REAL;
	PI_AlarmLowLimit : REAL;
	PI_AlarmLowLowLimit : REAL;
	
	PI_AlarmDelay_HH : LREAL;
	PI_AlarmDelay_H : LREAL;
	PI_AlarmDelay_L : LREAL;
	PI_AlarmDelay_LL : LREAL;
	
	Alarm_Ack_HH : BOOL;
	Alarm_Ack_H : BOOL;
	Alarm_Ack_L : BOOL;
	Alarm_Ack_LL : BOOL;
	
	PI_Interlock : BOOL;
	
	ENABLE_SCALING : BOOL;
	PI_PV_MAX_IN : INT;
	PI_PV_MIN_IN : INT;
	PI_PV_MAX_OUT : INT;
	PI_PV_MIN_OUT : INT;
END_VAR
VAR_OUTPUT
	
	PO_AUTO_ON :BOOL;
	PO_MANUAL_ON : BOOL;
	PO_HMI_HAND_ON : BOOL;
	
	PO_OUT_ON : BOOL;
	PO_OUT_OFF :BOOL;
	
	PO_Interlocked : BOOL;
	
	PO_PV_SCALED : REAL;
	
	PO_ALARM_HH : BOOL;
	PO_ALARM_H : BOOL;
	PO_ALARM_L : BOOL;
	PO_ALARM_LL : BOOL;
END_VAR
VAR_IN_OUT
	
END_VAR
VAR
	SR_Auto: SR;
	SR_Manual : SR;
	
	Alarm_limit_Exceeded_HH : BOOL;
	Alarm_limit_Exceeded_H : BOOL;
	Alarm_limit_Exceeded_L : BOOL;
	Alarm_limit_Exceeded_LL : BOOL;
	
	alarmDelay_HH : systemTimeDelay;
	alarmDelay_H : systemTimeDelay;
	alarmDelay_L : systemTimeDelay;
	alarmDelay_LL : systemTimeDelay;
	
	DelayForHistorianBit_HH: TON;
	DelayForHistorianBit_H: TON;
	DelayForHistorianBit_L: TON;
	DelayForHistorianBit_LL: TON;
	
	HistorianBit_HH :BOOL;
	HistorianBit_H :BOOL;
	HistorianBit_L :BOOL;
	HistorianBit_LL :BOOL;
	
	MODE_HANDLER : FB_MODE_HANDLER;
	
	scale : Tc2_ControllerToolbox.FB_CTRL_SCALE;
	scaleParams : ST_CTRL_SCALE_PARAMS;
	
	MODEHANDLER_AUTO_ON : BOOL;
	MODEHANDLER_MANUAL_ON : BOOL;
END_VAR

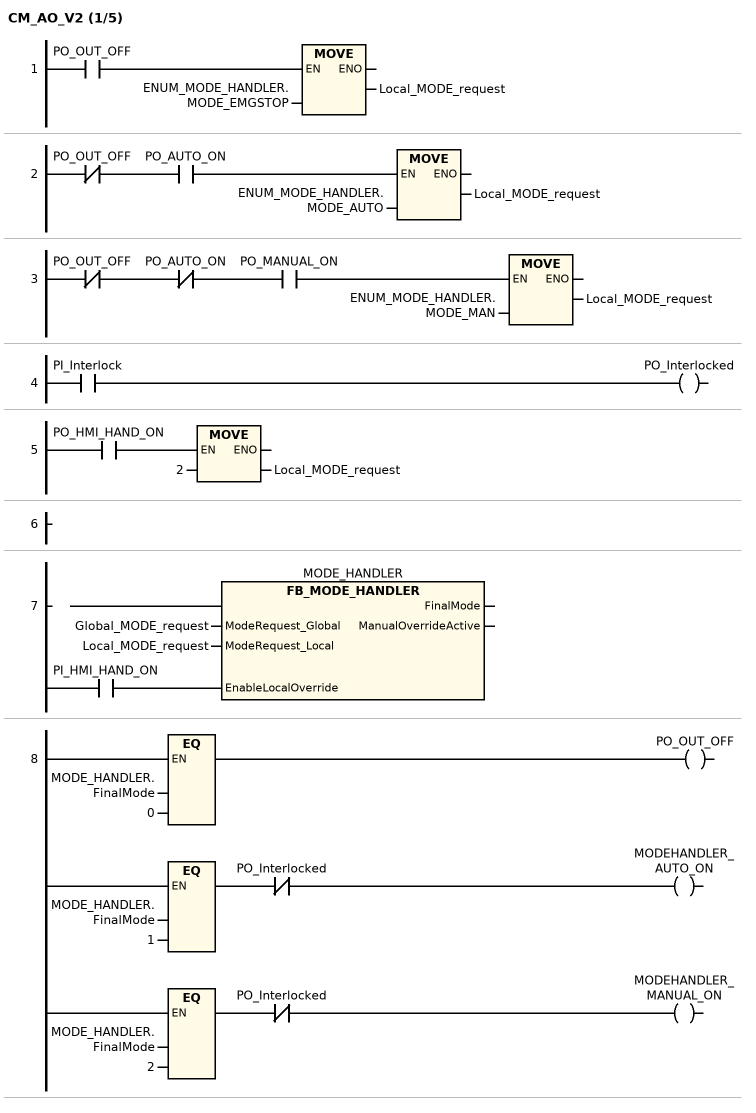
// NETWORK 1
IF PO_OUT_OFF THEN Local_MODE_request := ENUM_MODE_HANDLER.MODE_EMGSTOP; END_IF

// NETWORK 2
IF NOT PO_OUT_OFF AND PO_AUTO_ON THEN Local_MODE_request := ENUM_MODE_HANDLER.MODE_AUTO; END_IF

// NETWORK 3
IF NOT PO_OUT_OFF AND NOT PO_AUTO_ON AND PO_MANUAL_ON THEN Local_MODE_request := ENUM_MODE_HANDLER.MODE_MAN; END_IF

// NETWORK 4
PO_Interlocked := PI_Interlock;

// NETWORK 5
IF PO_HMI_HAND_ON THEN Local_MODE_request := 2; END_IF

// NETWORK 6

// NETWORK 7
MODE_HANDLER(
    ModeRequest_Global := Global_MODE_request,
    ModeRequest_Local := Local_MODE_request,
    EnableLocalOverride := PI_HMI_HAND_ON); // FB_MODE_HANDLER

// NETWORK 8
PO_OUT_OFF := MODE_HANDLER.FinalMode = 0;
MODEHANDLER_AUTO_ON := MODE_HANDLER.FinalMode = 1 AND NOT PO_Interlocked;
MODEHANDLER_MANUAL_ON := MODE_HANDLER.FinalMode = 2 AND NOT PO_Interlocked;

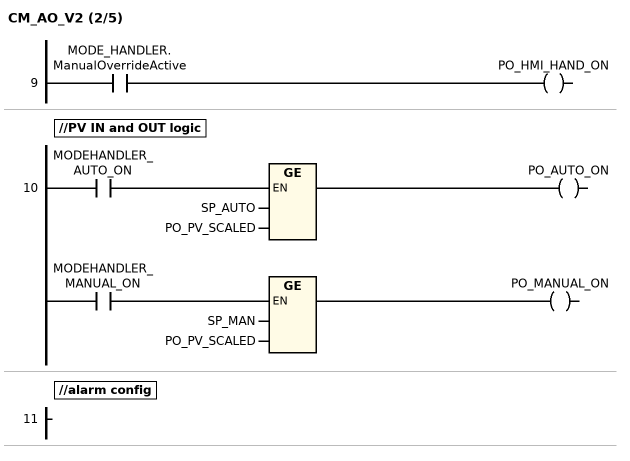
// NETWORK 9
PO_HMI_HAND_ON := MODE_HANDLER.ManualOverrideActive;

// NETWORK 10
// label: //PV IN and OUT logic
PO_AUTO_ON := MODEHANDLER_AUTO_ON AND SP_AUTO >= PO_PV_SCALED;
PO_MANUAL_ON := MODEHANDLER_MANUAL_ON AND SP_MAN >= PO_PV_SCALED;

// NETWORK 11
// label: //alarm config

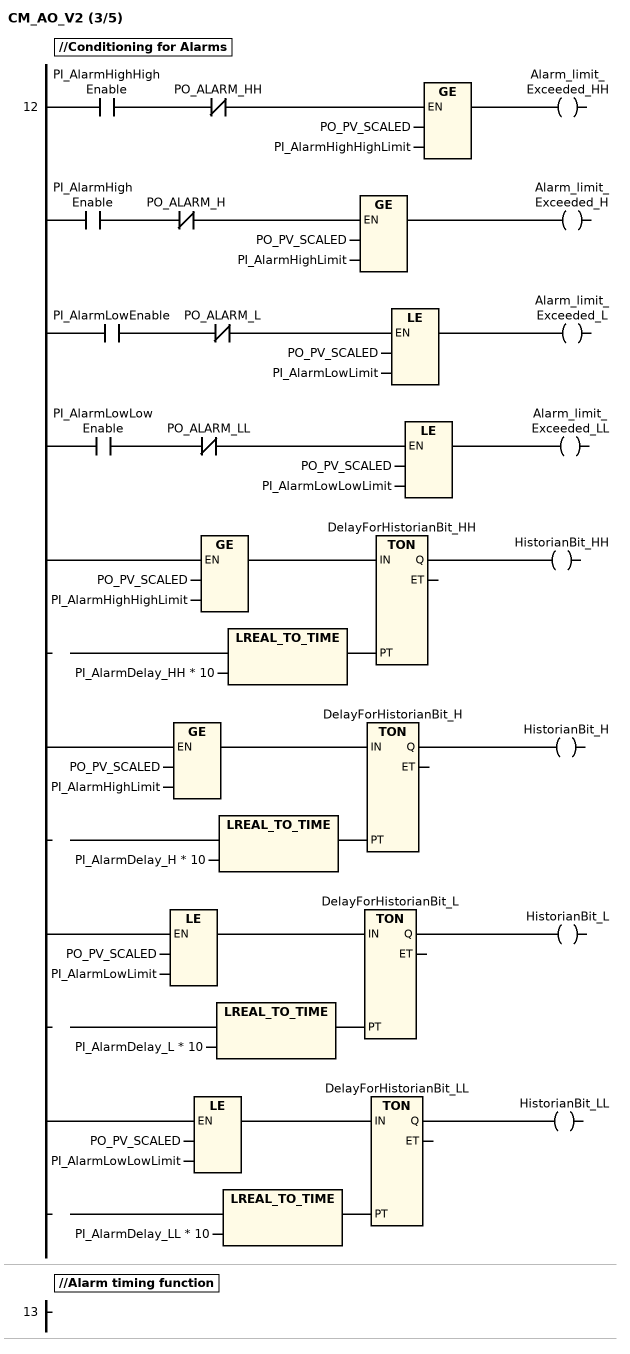
// NETWORK 12
// label: //Conditioning for Alarms
Alarm_limit_Exceeded_HH := PI_AlarmHighHighEnable AND NOT PO_ALARM_HH AND PO_PV_SCALED >= PI_AlarmHighHighLimit;
Alarm_limit_Exceeded_H := PI_AlarmHighEnable AND NOT PO_ALARM_H AND PO_PV_SCALED >= PI_AlarmHighLimit;
Alarm_limit_Exceeded_L := PI_AlarmLowEnable AND NOT PO_ALARM_L AND PO_PV_SCALED <= PI_AlarmLowLimit;
Alarm_limit_Exceeded_LL := PI_AlarmLowLowEnable AND NOT PO_ALARM_LL AND PO_PV_SCALED <= PI_AlarmLowLowLimit;
DelayForHistorianBit_HH(IN := PO_PV_SCALED >= PI_AlarmHighHighLimit, PT := LREAL_TO_TIME(PI_AlarmDelay_HH * 10)); // TON
HistorianBit_HH := DelayForHistorianBit_HH.Q;
DelayForHistorianBit_H(IN := PO_PV_SCALED >= PI_AlarmHighLimit, PT := LREAL_TO_TIME(PI_AlarmDelay_H * 10)); // TON
HistorianBit_H := DelayForHistorianBit_H.Q;
DelayForHistorianBit_L(IN := PO_PV_SCALED <= PI_AlarmLowLimit, PT := LREAL_TO_TIME(PI_AlarmDelay_L * 10)); // TON
HistorianBit_L := DelayForHistorianBit_L.Q;
DelayForHistorianBit_LL(IN := PO_PV_SCALED <= PI_AlarmLowLowLimit, PT := LREAL_TO_TIME(PI_AlarmDelay_LL * 10)); // TON
HistorianBit_LL := DelayForHistorianBit_LL.Q;

// NETWORK 13
// label: //Alarm timing function

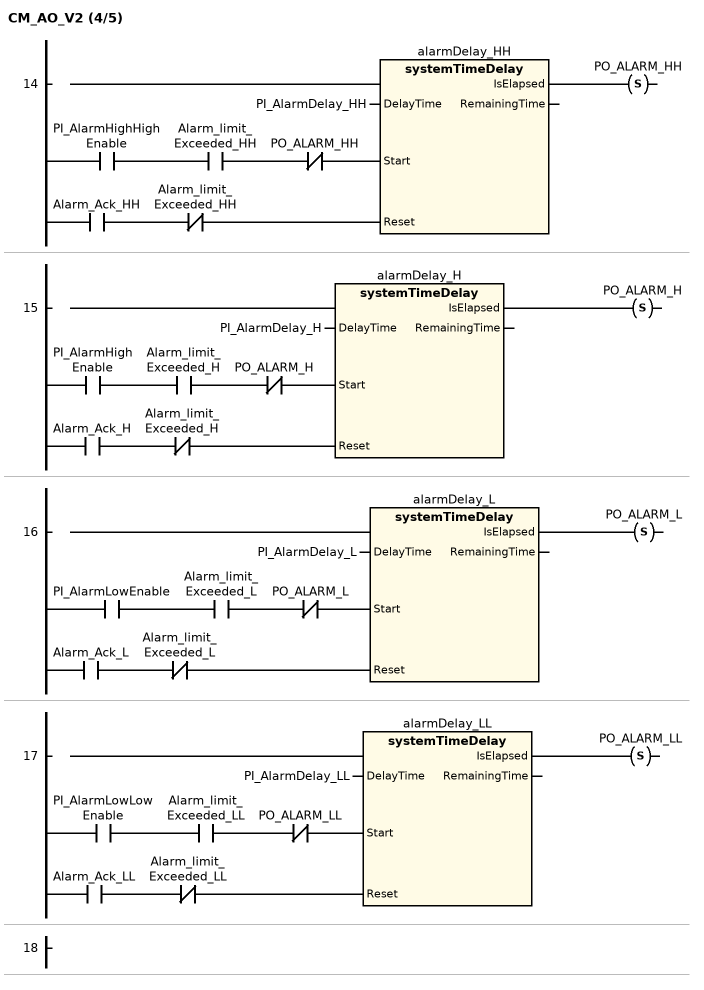
// NETWORK 14
alarmDelay_HH(
    DelayTime := PI_AlarmDelay_HH,
    Start := PI_AlarmHighHighEnable AND Alarm_limit_Exceeded_HH AND NOT PO_ALARM_HH,
    Reset := Alarm_Ack_HH AND NOT Alarm_limit_Exceeded_HH); // systemTimeDelay
PO_ALARM_HH S= alarmDelay_HH.IsElapsed;

// NETWORK 15
alarmDelay_H(
    DelayTime := PI_AlarmDelay_H,
    Start := PI_AlarmHighEnable AND Alarm_limit_Exceeded_H AND NOT PO_ALARM_H,
    Reset := Alarm_Ack_H AND NOT Alarm_limit_Exceeded_H); // systemTimeDelay
PO_ALARM_H S= alarmDelay_H.IsElapsed;

// NETWORK 16
alarmDelay_L(
    DelayTime := PI_AlarmDelay_L,
    Start := PI_AlarmLowEnable AND Alarm_limit_Exceeded_L AND NOT PO_ALARM_L,
    Reset := Alarm_Ack_L AND NOT Alarm_limit_Exceeded_L); // systemTimeDelay
PO_ALARM_L S= alarmDelay_L.IsElapsed;

// NETWORK 17
alarmDelay_LL(
    DelayTime := PI_AlarmDelay_LL,
    Start := PI_AlarmLowLowEnable AND Alarm_limit_Exceeded_LL AND NOT PO_ALARM_LL,
    Reset := Alarm_Ack_LL AND NOT Alarm_limit_Exceeded_LL); // systemTimeDelay
PO_ALARM_LL S= alarmDelay_LL.IsElapsed;

// NETWORK 18

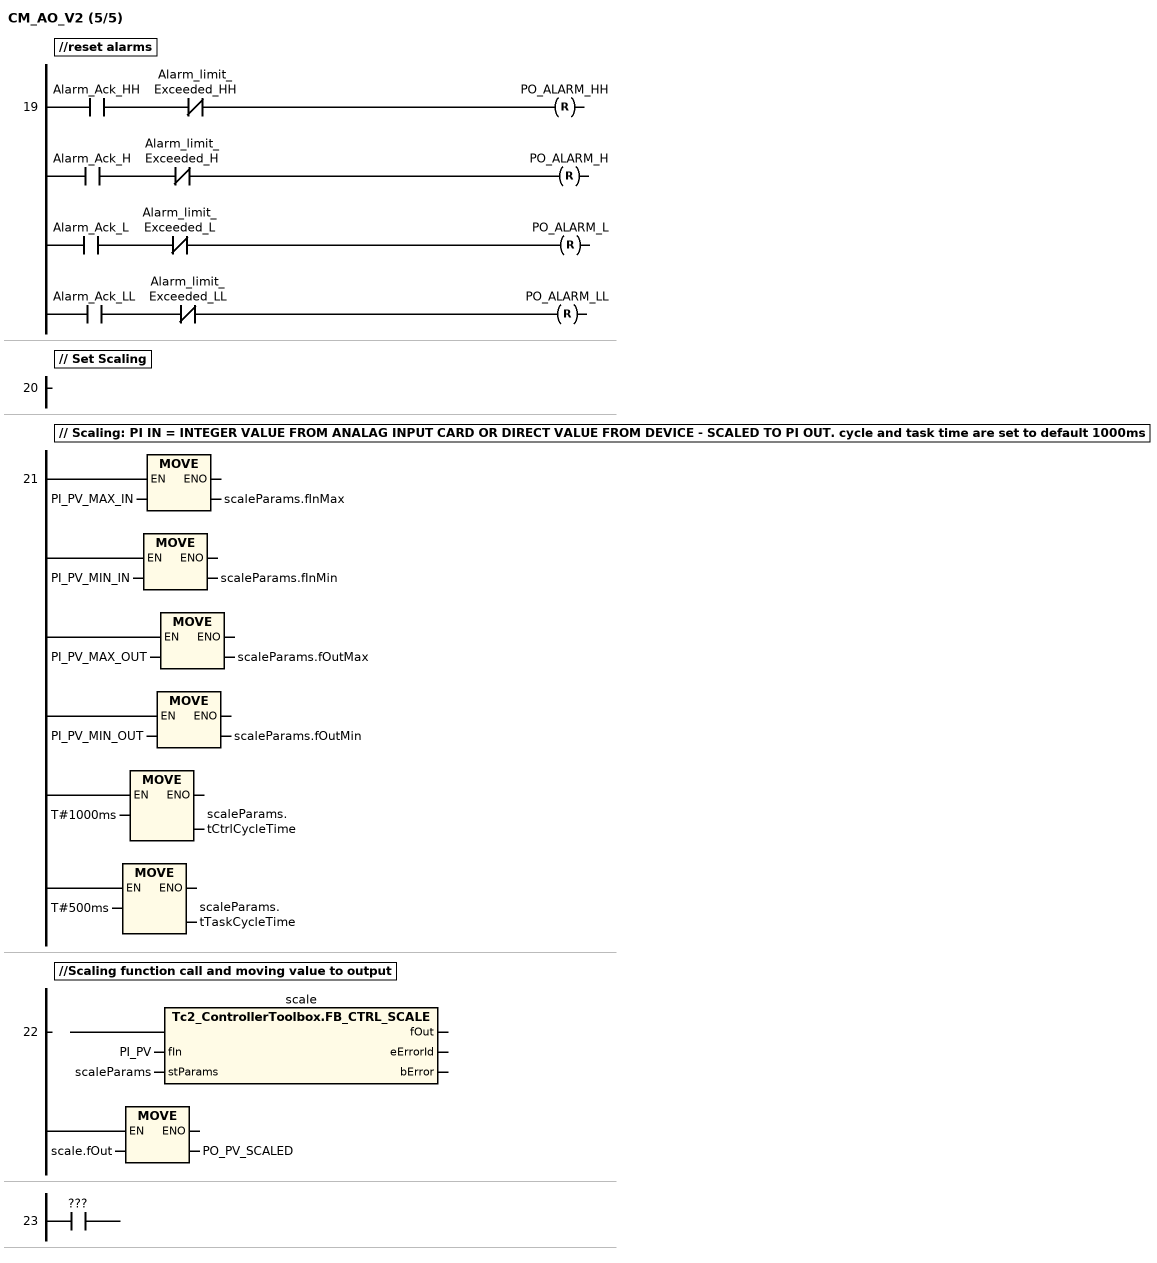
// NETWORK 19
// label: //reset alarms
PO_ALARM_HH R= Alarm_Ack_HH AND NOT Alarm_limit_Exceeded_HH;
PO_ALARM_H R= Alarm_Ack_H AND NOT Alarm_limit_Exceeded_H;
PO_ALARM_L R= Alarm_Ack_L AND NOT Alarm_limit_Exceeded_L;
PO_ALARM_LL R= Alarm_Ack_LL AND NOT Alarm_limit_Exceeded_LL;

// NETWORK 20
// label: // Set Scaling

// NETWORK 21
// label: // Scaling: PI IN = INTEGER VALUE FROM ANALAG INPUT CARD OR DIRECT VALUE FROM DEVICE - SCALED TO PI OUT. cycle and task time are set to default 1000ms
scaleParams.fInMax := PI_PV_MAX_IN;
scaleParams.fInMin := PI_PV_MIN_IN;
scaleParams.fOutMax := PI_PV_MAX_OUT;
scaleParams.fOutMin := PI_PV_MIN_OUT;
scaleParams.tCtrlCycleTime := T#1000ms;
scaleParams.tTaskCycleTime := T#500ms;

// NETWORK 22
// label: //Scaling function call and moving value to output
scale(fIn := PI_PV, stParams := scaleParams); // Tc2_ControllerToolbox.FB_CTRL_SCALE
PO_PV_SCALED := scale.fOut;

// NETWORK 23

END_FUNCTION_BLOCK

// ---- POUs/CM_V2/CM_Sensor2State_V2.TcPOU
FUNCTION_BLOCK CM_Sensor2State_V2
VAR_INPUT
	PI_ManualMode : BOOL;
	PI_AutoMode : BOOL;
	
	PI_HMI_HAND : BOOL;
	PI_HMI_HAND_ON : BOOL;
	
	PI_Manual_ON : BOOL;
	PI_AutoHigh : BOOL;
	
	PI_AlarmHighEnable : BOOL;
	PI_AlarmLowEnable : BOOL;
	PI_Alarmdelay_H : DINT;
	PI_Alarmdelay_L : DINT;
	
	PI_Alarm_Condition_H : BOOL;
	PI_Alarm_Condition_L : BOOL;
	
	
	
END_VAR
VAR_OUTPUT
	PO_HMI_HAND : BOOL;
	PO_Manual : BOOL;
	PO_High : BOOL;
	
	PO_Alarm_H : BOOL;
	PO_Alarm_L : BOOL;
END_VAR
VAR
	Alarm_limit_Exceeded_H : BOOL;
	Alarm_limit_Exceeded_L : BOOL;
	
	prg_scan_H : DINT; // used for alarm delay
	prg_scan_L : DINT; // used for alarm delay
	
	Alarm_Ack_H : BOOL;
	Alarm_Ack_L : BOOL;
	
	alarmDelay_H : systemTimeDelay;
	alarmDelay_L : systemTimeDelay;
	
	DelayForHistorianBit_H: TON;
	DelayForHistorianBit_L: TON;
END_VAR
VAR_IN_OUT
	CM_UDT_CTRL : Udt_CM_Sensor2State;
	Plant_control : Udt_PlantControl;
END_VAR

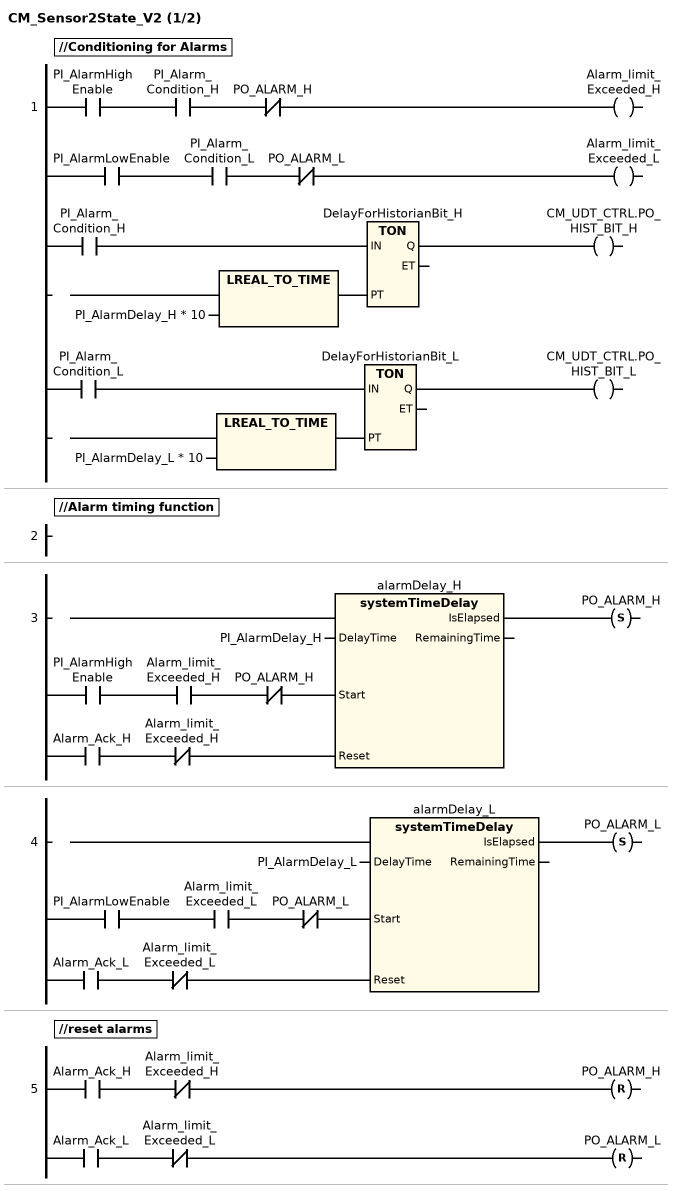
// NETWORK 1
// label: //Conditioning for Alarms
Alarm_limit_Exceeded_H := PI_AlarmHighEnable AND PI_Alarm_Condition_H AND NOT PO_ALARM_H;
Alarm_limit_Exceeded_L := PI_AlarmLowEnable AND PI_Alarm_Condition_L AND NOT PO_ALARM_L;
DelayForHistorianBit_H(IN := PI_Alarm_Condition_H, PT := LREAL_TO_TIME(PI_AlarmDelay_H * 10)); // TON
CM_UDT_CTRL.PO_HIST_BIT_H := DelayForHistorianBit_H.Q;
DelayForHistorianBit_L(IN := PI_Alarm_Condition_L, PT := LREAL_TO_TIME(PI_AlarmDelay_L * 10)); // TON
CM_UDT_CTRL.PO_HIST_BIT_L := DelayForHistorianBit_L.Q;

// NETWORK 2
// label: //Alarm timing function

// NETWORK 3
alarmDelay_H(
    DelayTime := PI_AlarmDelay_H,
    Start := PI_AlarmHighEnable AND Alarm_limit_Exceeded_H AND NOT PO_ALARM_H,
    Reset := Alarm_Ack_H AND NOT Alarm_limit_Exceeded_H); // systemTimeDelay
PO_ALARM_H S= alarmDelay_H.IsElapsed;

// NETWORK 4
alarmDelay_L(
    DelayTime := PI_AlarmDelay_L,
    Start := PI_AlarmLowEnable AND Alarm_limit_Exceeded_L AND NOT PO_ALARM_L,
    Reset := Alarm_Ack_L AND NOT Alarm_limit_Exceeded_L); // systemTimeDelay
PO_ALARM_L S= alarmDelay_L.IsElapsed;

// NETWORK 5
// label: //reset alarms
PO_ALARM_H R= Alarm_Ack_H AND NOT Alarm_limit_Exceeded_H;
PO_ALARM_L R= Alarm_Ack_L AND NOT Alarm_limit_Exceeded_L;

